LIN {X 0,Y 447.566,Z 552.365,A -85,B 0,C 180,E1 -8885.391,E2 -8885.391} C_VEL
LIN {X 0,Y 445.234,Z 544.551,A -85,B 0,C 180,E1 -8886.114,E2 -8886.114} C_VEL
LIN {X 0,Y 442.806,Z 536.367,A -85,B 0,C 180,E1 -8886.763,E2 -8886.763} C_VEL
LIN {X 0,Y 442.293,Z 531.074,A -85,B 0,C 180,E1 -8887.095,E2 -8887.095} C_VEL
LIN {X 0,Y 442.72,Z 518.254,A -85,B 0,C 180,E1 -8887.696,E2 -8887.696} C_VEL
LIN {X 0,Y 443.107,Z 504.32,A -85,B 0,C 180,E1 -8888.13,E2 -8888.13} C_VEL
LIN {X 0,Y 444.089,Z 414.582,A -85,B 0,C 180,E1 -8889.651,E2 -8889.651} C_VEL
LIN {X 0,Y 440.694,Z 396.943,A -85,B 0,C 180,E1 -8890.111,E2 -8890.111} C_VEL
LIN {X 0,Y 441.167,Z 386.817,A -85,B 0,C 180,E1 -8892.38,E2 -8892.38} C_VEL
LIN {X 0,Y 439.924,Z 378.992,A -85,B 0,C 180,E1 -8894.24,E2 -8894.24} C_VEL
LIN {X 0,Y 439.488,Z 376.743,A -85,B 0,C 180,E1 -8894.819,E2 -8894.819} C_VEL
LIN {X 0,Y 439.491,Z 376.739,A -85,B 0,C 180,E1 -8898,E2 -8898} C_VEL
LIN {X 0,Y 439.538,Z 376.73,A -85,B 0,C 180,E1 -8901.725,E2 -8901.725} C_VEL
LIN {X 0,Y 439.615,Z 376.728,A -85,B 0,C 180,E1 -8904.495,E2 -8904.495} C_VEL
LIN {X 0,Y 439.639,Z 376.722,A -85,B 0,C 180,E1 -8908.167,E2 -8908.167} C_VEL
LIN {X 0,Y 439.767,Z 376.705,A -85,B 0,C 180,E1 -8909.999,E2 -8909.999} C_VEL
LIN {X 0,Y 439.659,Z 376.717,A -85,B 0,C 180,E1 -8912.747,E2 -8912.747} C_VEL
LIN {X 0,Y 439.621,Z 376.724,A -85,B 0,C 180,E1 -8916.424,E2 -8916.424} C_VEL
LIN {X 0,Y 439.501,Z 376.734,A -85,B 0,C 180,E1 -8919.2,E2 -8919.2} C_VEL
LIN {X 0,Y 439.467,Z 376.739,A -85,B 0,C 180,E1 -8922.936,E2 -8922.936} C_VEL
LIN {X 0,Y 439.461,Z 376.743,A -85,B 0,C 180,E1 -8926.353,E2 -8926.353} C_VEL
LIN {X 0,Y 439.403,Z 376.75,A -85,B 0,C 180,E1 -8929.625,E2 -8929.625} C_VEL
LIN {X 0,Y 439.363,Z 376.753,A -85,B 0,C 180,E1 -8932.574,E2 -8932.574} C_VEL
LIN {X 0,Y 439.396,Z 376.752,A -85,B 0,C 180,E1 -8935.584,E2 -8935.584} C_VEL
LIN {X 0,Y 439.423,Z 376.744,A -85,B 0,C 180,E1 -8938.671,E2 -8938.671} C_VEL
LIN {X 0,Y 439.38,Z 376.753,A -85,B 0,C 180,E1 -8942.032,E2 -8942.032} C_VEL
LIN {X 0,Y 439.393,Z 376.752,A -85,B 0,C 180,E1 -8945.339,E2 -8945.339} C_VEL
LIN {X 0,Y 439.394,Z 376.748,A -85,B 0,C 180,E1 -8948.592,E2 -8948.592} C_VEL
LIN {X 0,Y 439.394,Z 376.752,A -85,B 0,C 180,E1 -8951.257,E2 -8951.257} C_VEL
LIN {X 0,Y 439.4,Z 376.751,A -85,B 0,C 180,E1 -8954.727,E2 -8954.727} C_VEL
LIN {X 0,Y 439.447,Z 376.896,A -85,B 0,C 180,E1 -8956.182,E2 -8956.182} C_VEL
LIN {X 0,Y 440.645,Z 383.573,A -85,B 0,C 180,E1 -8957.581,E2 -8957.581} C_VEL
LIN {X 0,Y 440.586,Z 391.432,A -85,B 0,C 180,E1 -8959.155,E2 -8959.155} C_VEL
LIN {X 0,Y 440.543,Z 396.061,A -85,B 0,C 180,E1 -8960.073,E2 -8960.073} C_VEL
LIN {X 0,Y 443.892,Z 415.086,A -85,B 0,C 180,E1 -8960.552,E2 -8960.552} C_VEL
LIN {X 0,Y 442.71,Z 504.451,A -85,B 0,C 180,E1 -8962.148,E2 -8962.148} C_VEL
LIN {X 0,Y 442.406,Z 517.033,A -85,B 0,C 180,E1 -8962.539,E2 -8962.539} C_VEL
LIN {X 0,Y 441.999,Z 529.5,A -85,B 0,C 180,E1 -8963.112,E2 -8963.112} C_VEL
LIN {X 0,Y 441.424,Z 542.347,A -85,B 0,C 180,E1 -8963.908,E2 -8963.908} C_VEL
LIN {X 0,Y 440.846,Z 554.105,A -85,B 0,C 180,E1 -8964.864,E2 -8964.864} C_VEL
LIN {X 0,Y 440.299,Z 564.276,A -85,B 0,C 180,E1 -8965.898,E2 -8965.898} C_VEL
LIN {X 0,Y 439.735,Z 573.76,A -85,B 0,C 180,E1 -8967.084,E2 -8967.084} C_VEL
LIN {X 0,Y 439.346,Z 582.271,A -85,B 0,C 180,E1 -8968.406,E2 -8968.406} C_VEL
LIN {X 0,Y 438.905,Z 589.744,A -85,B 0,C 180,E1 -8969.843,E2 -8969.843} C_VEL
LIN {X 0,Y 438.641,Z 595.595,A -85,B 0,C 180,E1 -8971.271,E2 -8971.271} C_VEL
LIN {X 0,Y 438.411,Z 600.454,A -85,B 0,C 180,E1 -8972.814,E2 -8972.814} C_VEL
LIN {X 0,Y 438.281,Z 603.953,A -85,B 0,C 180,E1 -8974.345,E2 -8974.345} C_VEL
LIN {X 0,Y 438.161,Z 606.47,A -85,B 0,C 180,E1 -8976.098,E2 -8976.098} C_VEL
LIN {X 0,Y 438.109,Z 607.349,A -85,B 0,C 180,E1 -8977.356,E2 -8977.356} C_VEL
LIN {X 0,Y 438.125,Z 607.446,A -85,B 0,C 180,E1 -8978.49,E2 -8978.49} C_VEL
LIN {X 0,Y 438.167,Z 607.132,A -85,B 0,C 180,E1 -8979.337,E2 -8979.337} C_VEL
LIN {X 0,Y 438.189,Z 606.343,A -85,B 0,C 180,E1 -8980.317,E2 -8980.317} C_VEL
LIN {X 0,Y 438.258,Z 605.052,A -85,B 0,C 180,E1 -8981.293,E2 -8981.293} C_VEL
LIN {X 0,Y 438.387,Z 602.262,A -85,B 0,C 180,E1 -8982.747,E2 -8982.747} C_VEL
LIN {X 0,Y 438.537,Z 598.37,A -85,B 0,C 180,E1 -8984.19,E2 -8984.19} C_VEL
LIN {X 0,Y 438.814,Z 593.262,A -85,B 0,C 180,E1 -8985.626,E2 -8985.626} C_VEL
LIN {X 0,Y 439.199,Z 586.765,A -85,B 0,C 180,E1 -8987.054,E2 -8987.054} C_VEL
LIN {X 0,Y 439.664,Z 578.655,A -85,B 0,C 180,E1 -8988.474,E2 -8988.474} C_VEL
LIN {X 0,Y 440.14,Z 570.383,A -85,B 0,C 180,E1 -8989.651,E2 -8989.651} C_VEL
LIN {X 0,Y 440.783,Z 560.176,A -85,B 0,C 180,E1 -8990.825,E2 -8990.825} C_VEL
LIN {X 0,Y 441.464,Z 548.726,A -85,B 0,C 180,E1 -8991.878,E2 -8991.878} C_VEL
LIN {X 0,Y 442.006,Z 537.482,A -85,B 0,C 180,E1 -8992.692,E2 -8992.692} C_VEL
LIN {X 0,Y 442.484,Z 524.938,A -85,B 0,C 180,E1 -8993.387,E2 -8993.387} C_VEL
LIN {X 0,Y 442.894,Z 511.882,A -85,B 0,C 180,E1 -8993.908,E2 -8993.908} C_VEL
LIN {X 0,Y 443.187,Z 497.848,A -85,B 0,C 180,E1 -8994.255,E2 -8994.255} C_VEL
LIN {X 0,Y 444.33,Z 414.224,A -85,B 0,C 180,E1 -8995.784,E2 -8995.784} C_VEL
LIN {X 0,Y 440.81,Z 396.654,A -85,B 0,C 180,E1 -8996.308,E2 -8996.308} C_VEL
LIN {X 0,Y 441.009,Z 384.795,A -85,B 0,C 180,E1 -8998.63,E2 -8998.63} C_VEL
LIN {X 0,Y 439.724,Z 376.714,A -85,B 0,C 180,E1 -9000.286,E2 -9000.286} C_VEL
LIN {X 0,Y 439.647,Z 376.725,A -85,B 0,C 180,E1 -9002.749,E2 -9002.749} C_VEL
LIN {X 0,Y 439.608,Z 376.728,A -85,B 0,C 180,E1 -9006.425,E2 -9006.425} C_VEL
LIN {X 0,Y 439.491,Z 376.739,A -85,B 0,C 180,E1 -9009.202,E2 -9009.202} C_VEL
LIN {X 0,Y 439.493,Z 376.741,A -85,B 0,C 180,E1 -9012.727,E2 -9012.727} C_VEL
LIN {X 0,Y 439.449,Z 376.747,A -85,B 0,C 180,E1 -9016.355,E2 -9016.355} C_VEL
LIN {X 0,Y 439.425,Z 376.75,A -85,B 0,C 180,E1 -9019.625,E2 -9019.625} C_VEL
LIN {X 0,Y 439.376,Z 376.752,A -85,B 0,C 180,E1 -9022.575,E2 -9022.575} C_VEL
LIN {X 0,Y 439.405,Z 376.753,A -85,B 0,C 180,E1 -9025.585,E2 -9025.585} C_VEL
LIN {X 0,Y 439.415,Z 376.747,A -85,B 0,C 180,E1 -9028.674,E2 -9028.674} C_VEL
LIN {X 0,Y 439.374,Z 376.755,A -85,B 0,C 180,E1 -9032.034,E2 -9032.034} C_VEL
LIN {X 0,Y 439.387,Z 376.754,A -85,B 0,C 180,E1 -9035.342,E2 -9035.342} C_VEL
LIN {X 0,Y 439.382,Z 376.751,A -85,B 0,C 180,E1 -9038.595,E2 -9038.595} C_VEL
LIN {X 0,Y 439.382,Z 376.755,A -85,B 0,C 180,E1 -9041.258,E2 -9041.258} C_VEL
LIN {X 0,Y 439.399,Z 376.75,A -85,B 0,C 180,E1 -9044.73,E2 -9044.73} C_VEL
LIN {X 0,Y 439.391,Z 376.751,A -85,B 0,C 180,E1 -9047.797,E2 -9047.797} C_VEL
LIN {X 0,Y 439.424,Z 376.746,A -85,B 0,C 180,E1 -9050.229,E2 -9050.229} C_VEL
LIN {X 0,Y 439.372,Z 376.753,A -85,B 0,C 180,E1 -9053.715,E2 -9053.715} C_VEL
LIN {X 0,Y 439.372,Z 376.758,A -85,B 0,C 180,E1 -9057.056,E2 -9057.056} C_VEL
LIN {X 0,Y 439.395,Z 376.753,A -85,B 0,C 180,E1 -9060.277,E2 -9060.277} C_VEL
LIN {X 0,Y 439.481,Z 376.95,A -85,B 0,C 180,E1 -9063.401,E2 -9063.401} C_VEL
LIN {X 0,Y 441.912,Z 389.672,A -85,B 0,C 180,E1 -9066.076,E2 -9066.076} C_VEL
LIN {X 0,Y 441.931,Z 394.416,A -85,B 0,C 180,E1 -9067.01,E2 -9067.01} C_VEL
LIN {X 0,Y 440.88,Z 413.613,A -85,B 0,C 180,E1 -9070.686,E2 -9070.686} C_VEL
LIN {X 0,Y 440.489,Z 420.151,A -85,B 0,C 180,E1 -9071.923,E2 -9071.923} C_VEL
LIN {X 0,Y 443.955,Z 442.221,A -85,B 0,C 180,E1 -9072.443,E2 -9072.443} C_VEL
LIN {X 0,Y 443.036,Z 528.918,A -85,B 0,C 180,E1 -9073.913,E2 -9073.913} C_VEL
LIN {X 0,Y 442.567,Z 542.639,A -85,B 0,C 180,E1 -9074.339,E2 -9074.339} C_VEL
LIN {X 0,Y 442.07,Z 555.017,A -85,B 0,C 180,E1 -9074.912,E2 -9074.912} C_VEL
LIN {X 0,Y 441.505,Z 566.099,A -85,B 0,C 180,E1 -9075.599,E2 -9075.599} C_VEL
LIN {X 0,Y 440.859,Z 577.655,A -85,B 0,C 180,E1 -9076.517,E2 -9076.517} C_VEL
LIN {X 0,Y 440.298,Z 588.106,A -85,B 0,C 180,E1 -9077.557,E2 -9077.557} C_VEL
LIN {X 0,Y 439.725,Z 597.48,A -85,B 0,C 180,E1 -9078.711,E2 -9078.711} C_VEL
LIN {X 0,Y 439.182,Z 606.551,A -85,B 0,C 180,E1 -9080.096,E2 -9080.096} C_VEL
LIN {X 0,Y 438.798,Z 613.859,A -85,B 0,C 180,E1 -9081.481,E2 -9081.481} C_VEL
LIN {X 0,Y 438.582,Z 618.796,A -85,B 0,C 180,E1 -9082.636,E2 -9082.636} C_VEL
LIN {X 0,Y 438.384,Z 623.457,A -85,B 0,C 180,E1 -9083.978,E2 -9083.978} C_VEL
LIN {X 0,Y 438.341,Z 627.253,A -85,B 0,C 180,E1 -9085.403,E2 -9085.403} C_VEL
LIN {X 0,Y 438.28,Z 629.143,A -85,B 0,C 180,E1 -9086.324,E2 -9086.324} C_VEL
LIN {X 0,Y 438.34,Z 630.568,A -85,B 0,C 180,E1 -9087.244,E2 -9087.244} C_VEL
LIN {X 0,Y 438.252,Z 632.191,A -85,B 0,C 180,E1 -9089.082,E2 -9089.082} C_VEL
LIN {X 0,Y 438.253,Z 632.415,A -85,B 0,C 180,E1 -9090.001,E2 -9090.001} C_VEL
LIN {X 0,Y 438.252,Z 632.202,A -85,B 0,C 180,E1 -9090.92,E2 -9090.92} C_VEL
LIN {X 0,Y 438.341,Z 630.585,A -85,B 0,C 180,E1 -9092.758,E2 -9092.758} C_VEL
LIN {X 0,Y 438.28,Z 629.174,A -85,B 0,C 180,E1 -9093.679,E2 -9093.679} C_VEL
LIN {X 0,Y 438.386,Z 626.213,A -85,B 0,C 180,E1 -9095.06,E2 -9095.06} C_VEL
LIN {X 0,Y 438.449,Z 622.202,A -85,B 0,C 180,E1 -9096.444,E2 -9096.444} C_VEL
LIN {X 0,Y 438.688,Z 616.038,A -85,B 0,C 180,E1 -9098.059,E2 -9098.059} C_VEL
LIN {X 0,Y 439.048,Z 609.304,A -85,B 0,C 180,E1 -9099.445,E2 -9099.445} C_VEL
LIN {X 0,Y 439.489,Z 600.961,A -85,B 0,C 180,E1 -9100.831,E2 -9100.831} C_VEL
LIN {X 0,Y 440.08,Z 592.405,A -85,B 0,C 180,E1 -9101.983,E2 -9101.983} C_VEL
LIN {X 0,Y 440.612,Z 582.48,A -85,B 0,C 180,E1 -9103.075,E2 -9103.075} C_VEL
LIN {X 0,Y 441.266,Z 571.393,A -85,B 0,C 180,E1 -9104.058,E2 -9104.058} C_VEL
LIN {X 0,Y 441.886,Z 559.936,A -85,B 0,C 180,E1 -9104.861,E2 -9104.861} C_VEL
LIN {X 0,Y 442.507,Z 548.123,A -85,B 0,C 180,E1 -9105.488,E2 -9105.488} C_VEL
LIN {X 0,Y 442.942,Z 535.462,A -85,B 0,C 180,E1 -9105.974,E2 -9105.974} C_VEL
LIN {X 0,Y 443.357,Z 522.565,A -85,B 0,C 180,E1 -9106.284,E2 -9106.284} C_VEL
LIN {X 0,Y 444.033,Z 441.38,A -85,B 0,C 180,E1 -9107.656,E2 -9107.656} C_VEL
LIN {X 0,Y 440.537,Z 419.596,A -85,B 0,C 180,E1 -9108.203,E2 -9108.203} C_VEL
LIN {X 0,Y 441.514,Z 402.491,A -85,B 0,C 180,E1 -9111.477,E2 -9111.477} C_VEL
LIN {X 0,Y 442.185,Z 391.264,A -85,B 0,C 180,E1 -9113.662,E2 -9113.662} C_VEL
LIN {X 0,Y 440.418,Z 381.325,A -85,B 0,C 180,E1 -9115.77,E2 -9115.77} C_VEL
LIN {X 0,Y 439.449,Z 376.748,A -85,B 0,C 180,E1 -9116.796,E2 -9116.796} C_VEL
LIN {X 0,Y 439.388,Z 376.757,A -85,B 0,C 180,E1 -9119.726,E2 -9119.726} C_VEL
LIN {X 0,Y 439.378,Z 376.757,A -85,B 0,C 180,E1 -9122.947,E2 -9122.947} C_VEL
LIN {X 0,Y 439.379,Z 376.754,A -85,B 0,C 180,E1 -9126.288,E2 -9126.288} C_VEL
LIN {X 0,Y 439.412,Z 376.751,A -85,B 0,C 180,E1 -9129.85,E2 -9129.85} C_VEL
LIN {X 0,Y 439.388,Z 376.755,A -85,B 0,C 180,E1 -9132.628,E2 -9132.628} C_VEL
LIN {X 0,Y 439.407,Z 376.753,A -85,B 0,C 180,E1 -9135.271,E2 -9135.271} C_VEL
LIN {X 0,Y 439.394,Z 376.755,A -85,B 0,C 180,E1 -9138.744,E2 -9138.744} C_VEL
LIN {X 0,Y 439.378,Z 376.752,A -85,B 0,C 180,E1 -9141.608,E2 -9141.608} C_VEL
LIN {X 0,Y 439.404,Z 376.752,A -85,B 0,C 180,E1 -9144.844,E2 -9144.844} C_VEL
LIN {X 0,Y 439.379,Z 376.752,A -85,B 0,C 180,E1 -9148.14,E2 -9148.14} C_VEL
LIN {X 0,Y 439.438,Z 376.743,A -85,B 0,C 180,E1 -9151.598,E2 -9151.598} C_VEL
LIN {X 0,Y 439.403,Z 376.749,A -85,B 0,C 180,E1 -9154.415,E2 -9154.415} C_VEL
LIN {X 0,Y 439.369,Z 376.747,A -85,B 0,C 180,E1 -9157.425,E2 -9157.425} C_VEL
LIN {X 0,Y 439.447,Z 376.742,A -85,B 0,C 180,E1 -9160.663,E2 -9160.663} C_VEL
LIN {X 0,Y 439.468,Z 376.745,A -85,B 0,C 180,E1 -9164.225,E2 -9164.225} C_VEL
LIN {X 0,Y 439.489,Z 376.741,A -85,B 0,C 180,E1 -9168.001,E2 -9168.001} C_VEL
LIN {X 0,Y 439.554,Z 376.731,A -85,B 0,C 180,E1 -9171.726,E2 -9171.726} C_VEL
LIN {X 0,Y 439.627,Z 376.724,A -85,B 0,C 180,E1 -9174.496,E2 -9174.496} C_VEL
LIN {X 0,Y 439.64,Z 376.723,A -85,B 0,C 180,E1 -9178.168,E2 -9178.168} C_VEL
LIN {X 0,Y 439.768,Z 376.706,A -85,B 0,C 180,E1 -9180,E2 -9180} C_VEL
LIN {X 0,Y 439.647,Z 376.718,A -85,B 0,C 180,E1 -9182.749,E2 -9182.749} C_VEL
LIN {X 0,Y 439.624,Z 376.721,A -85,B 0,C 180,E1 -9186.425,E2 -9186.425} C_VEL
LIN {X 0,Y 439.506,Z 376.736,A -85,B 0,C 180,E1 -9189.202,E2 -9189.202} C_VEL
LIN {X 0,Y 439.472,Z 376.74,A -85,B 0,C 180,E1 -9192.938,E2 -9192.938} C_VEL
LIN {X 0,Y 439.454,Z 376.744,A -85,B 0,C 180,E1 -9196.349,E2 -9196.349} C_VEL
LIN {X 0,Y 439.409,Z 376.753,A -85,B 0,C 180,E1 -9199.626,E2 -9199.626} C_VEL
LIN {X 0,Y 439.37,Z 376.754,A -85,B 0,C 180,E1 -9202.575,E2 -9202.575} C_VEL
LIN {X 0,Y 439.404,Z 376.752,A -85,B 0,C 180,E1 -9205.585,E2 -9205.585} C_VEL
LIN {X 0,Y 439.461,Z 376.78,A -85,B 0,C 180,E1 -9208.965,E2 -9208.965} C_VEL
LIN {X 0,Y 441.273,Z 386.843,A -85,B 0,C 180,E1 -9211.44,E2 -9211.44} C_VEL
LIN {X 0,Y 440.869,Z 397.525,A -85,B 0,C 180,E1 -9213.88,E2 -9213.88} C_VEL
LIN {X 0,Y 444.38,Z 415.736,A -85,B 0,C 180,E1 -9214.365,E2 -9214.365} C_VEL
LIN {X 0,Y 443.296,Z 504.669,A -85,B 0,C 180,E1 -9215.881,E2 -9215.881} C_VEL
LIN {X 0,Y 442.938,Z 517.91,A -85,B 0,C 180,E1 -9216.292,E2 -9216.292} C_VEL
LIN {X 0,Y 442.511,Z 529.911,A -85,B 0,C 180,E1 -9216.841,E2 -9216.841} C_VEL
LIN {X 0,Y 441.995,Z 541.351,A -85,B 0,C 180,E1 -9217.54,E2 -9217.54} C_VEL
LIN {X 0,Y 441.402,Z 552.126,A -85,B 0,C 180,E1 -9218.386,E2 -9218.386} C_VEL
LIN {X 0,Y 440.719,Z 563.511,A -85,B 0,C 180,E1 -9219.51,E2 -9219.51} C_VEL
LIN {X 0,Y 440.06,Z 572.934,A -85,B 0,C 180,E1 -9220.669,E2 -9220.669} C_VEL
LIN {X 0,Y 439.57,Z 581.346,A -85,B 0,C 180,E1 -9221.953,E2 -9221.953} C_VEL
LIN {X 0,Y 439.166,Z 587.526,A -85,B 0,C 180,E1 -9223.092,E2 -9223.092} C_VEL
LIN {X 0,Y 438.861,Z 593.327,A -85,B 0,C 180,E1 -9224.396,E2 -9224.396} C_VEL
LIN {X 0,Y 438.613,Z 598.01,A -85,B 0,C 180,E1 -9225.702,E2 -9225.702} C_VEL
LIN {X 0,Y 438.42,Z 601.693,A -85,B 0,C 180,E1 -9227.008,E2 -9227.008} C_VEL
LIN {X 0,Y 438.296,Z 604.387,A -85,B 0,C 180,E1 -9228.282,E2 -9228.282} C_VEL
LIN {X 0,Y 438.142,Z 606.786,A -85,B 0,C 180,E1 -9230.086,E2 -9230.086} C_VEL
LIN {X 0,Y 438.137,Z 607.642,A -85,B 0,C 180,E1 -9231.813,E2 -9231.813} C_VEL
LIN {X 0,Y 438.152,Z 607.06,A -85,B 0,C 180,E1 -9233.594,E2 -9233.594} C_VEL
LIN {X 0,Y 438.2,Z 605.696,A -85,B 0,C 180,E1 -9234.881,E2 -9234.881} C_VEL
LIN {X 0,Y 438.389,Z 602.878,A -85,B 0,C 180,E1 -9236.474,E2 -9236.474} C_VEL
LIN {X 0,Y 438.561,Z 598.488,A -85,B 0,C 180,E1 -9238.14,E2 -9238.14} C_VEL
LIN {X 0,Y 438.79,Z 593.541,A -85,B 0,C 180,E1 -9239.545,E2 -9239.545} C_VEL
LIN {X 0,Y 439.21,Z 586.801,A -85,B 0,C 180,E1 -9241.049,E2 -9241.049} C_VEL
LIN {X 0,Y 439.654,Z 579.288,A -85,B 0,C 180,E1 -9242.381,E2 -9242.381} C_VEL
LIN {X 0,Y 440.169,Z 570.074,A -85,B 0,C 180,E1 -9243.699,E2 -9243.699} C_VEL
LIN {X 0,Y 440.769,Z 560.449,A -85,B 0,C 180,E1 -9244.815,E2 -9244.815} C_VEL
LIN {X 0,Y 441.379,Z 550,A -85,B 0,C 180,E1 -9245.793,E2 -9245.793} C_VEL
LIN {X 0,Y 441.991,Z 538.279,A -85,B 0,C 180,E1 -9246.659,E2 -9246.659} C_VEL
LIN {X 0,Y 442.293,Z 531.074,A -85,B 0,C 180,E1 -9247.095,E2 -9247.095} C_VEL
LIN {X 0,Y 441.795,Z 525.662,A -85,B 0,C 180,E1 -9247.399,E2 -9247.399} C_VEL
LIN {X 0,Y 439.368,Z 516.782,A -85,B 0,C 180,E1 -9247.88,E2 -9247.88} C_VEL
LIN {X 0,Y 436.901,Z 507.688,A -85,B 0,C 180,E1 -9248.27,E2 -9248.27} C_VEL
LIN {X 0,Y 436.322,Z 501.949,A -85,B 0,C 180,E1 -9248.427,E2 -9248.427} C_VEL
LIN {X 0,Y 437.208,Z 415.029,A -85,B 0,C 180,E1 -9249.919,E2 -9249.919} C_VEL
LIN {X 0,Y 433.767,Z 397.177,A -85,B 0,C 180,E1 -9250.384,E2 -9250.384} C_VEL
LIN {X 0,Y 434.141,Z 387.363,A -85,B 0,C 180,E1 -9252.621,E2 -9252.621} C_VEL
LIN {X 0,Y 432.459,Z 377.619,A -85,B 0,C 180,E1 -9255.018,E2 -9255.018} C_VEL
LIN {X 0,Y 432.464,Z 377.614,A -85,B 0,C 180,E1 -9257.802,E2 -9257.802} C_VEL
LIN {X 0,Y 432.488,Z 377.608,A -85,B 0,C 180,E1 -9261.589,E2 -9261.589} C_VEL
LIN {X 0,Y 432.59,Z 377.603,A -85,B 0,C 180,E1 -9264.405,E2 -9264.405} C_VEL
LIN {X 0,Y 432.609,Z 377.598,A -85,B 0,C 180,E1 -9268.137,E2 -9268.137} C_VEL
LIN {X 0,Y 432.736,Z 377.581,A -85,B 0,C 180,E1 -9269.999,E2 -9269.999} C_VEL
LIN {X 0,Y 432.608,Z 377.595,A -85,B 0,C 180,E1 -9272.792,E2 -9272.792} C_VEL
LIN {X 0,Y 432.576,Z 377.601,A -85,B 0,C 180,E1 -9276.529,E2 -9276.529} C_VEL
LIN {X 0,Y 432.444,Z 377.614,A -85,B 0,C 180,E1 -9279.352,E2 -9279.352} C_VEL
LIN {X 0,Y 432.432,Z 377.616,A -85,B 0,C 180,E1 -9282.802,E2 -9282.802} C_VEL
LIN {X 0,Y 432.424,Z 377.618,A -85,B 0,C 180,E1 -9286.482,E2 -9286.482} C_VEL
LIN {X 0,Y 432.339,Z 377.634,A -85,B 0,C 180,E1 -9289.959,E2 -9289.959} C_VEL
LIN {X 0,Y 432.317,Z 377.63,A -85,B 0,C 180,E1 -9292.963,E2 -9292.963} C_VEL
LIN {X 0,Y 432.36,Z 377.629,A -85,B 0,C 180,E1 -9296.031,E2 -9296.031} C_VEL
LIN {X 0,Y 432.35,Z 377.627,A -85,B 0,C 180,E1 -9299.185,E2 -9299.185} C_VEL
LIN {X 0,Y 432.329,Z 377.629,A -85,B 0,C 180,E1 -9302.293,E2 -9302.293} C_VEL
LIN {X 0,Y 432.337,Z 377.627,A -85,B 0,C 180,E1 -9304.675,E2 -9304.675} C_VEL
LIN {X 0,Y 432.348,Z 377.627,A -85,B 0,C 180,E1 -9308.147,E2 -9308.147} C_VEL
LIN {X 0,Y 432.362,Z 377.631,A -85,B 0,C 180,E1 -9311.606,E2 -9311.606} C_VEL
LIN {X 0,Y 432.335,Z 377.631,A -85,B 0,C 180,E1 -9314.345,E2 -9314.345} C_VEL
LIN {X 0,Y 432.39,Z 377.751,A -85,B 0,C 180,E1 -9316.031,E2 -9316.031} C_VEL
LIN {X 0,Y 433.737,Z 385.68,A -85,B 0,C 180,E1 -9317.693,E2 -9317.693} C_VEL
LIN {X 0,Y 433.561,Z 396.365,A -85,B 0,C 180,E1 -9319.806,E2 -9319.806} C_VEL
LIN {X 0,Y 437.065,Z 415.855,A -85,B 0,C 180,E1 -9320.314,E2 -9320.314} C_VEL
LIN {X 0,Y 435.859,Z 503.979,A -85,B 0,C 180,E1 -9321.92,E2 -9321.92} C_VEL
LIN {X 0,Y 435.5,Z 517.172,A -85,B 0,C 180,E1 -9322.331,E2 -9322.331} C_VEL
LIN {X 0,Y 435.055,Z 529.986,A -85,B 0,C 180,E1 -9322.932,E2 -9322.932} C_VEL
LIN {X 0,Y 434.481,Z 542.469,A -85,B 0,C 180,E1 -9323.719,E2 -9323.719} C_VEL
LIN {X 0,Y 433.929,Z 553.476,A -85,B 0,C 180,E1 -9324.618,E2 -9324.618} C_VEL
LIN {X 0,Y 433.321,Z 563.929,A -85,B 0,C 180,E1 -9325.683,E2 -9325.683} C_VEL
LIN {X 0,Y 432.81,Z 572.642,A -85,B 0,C 180,E1 -9326.767,E2 -9326.767} C_VEL
LIN {X 0,Y 432.355,Z 581.436,A -85,B 0,C 180,E1 -9328.11,E2 -9328.11} C_VEL
LIN {X 0,Y 431.872,Z 589.21,A -85,B 0,C 180,E1 -9329.594,E2 -9329.594} C_VEL
LIN {X 0,Y 431.642,Z 594.154,A -85,B 0,C 180,E1 -9330.76,E2 -9330.76} C_VEL
LIN {X 0,Y 431.406,Z 599.473,A -85,B 0,C 180,E1 -9332.335,E2 -9332.335} C_VEL
LIN {X 0,Y 431.24,Z 603.332,A -85,B 0,C 180,E1 -9333.894,E2 -9333.894} C_VEL
LIN {X 0,Y 431.142,Z 605.168,A -85,B 0,C 180,E1 -9334.924,E2 -9334.924} C_VEL
LIN {X 0,Y 431.076,Z 606.522,A -85,B 0,C 180,E1 -9335.947,E2 -9335.947} C_VEL
LIN {X 0,Y 431.018,Z 607.322,A -85,B 0,C 180,E1 -9336.962,E2 -9336.962} C_VEL
LIN {X 0,Y 431.024,Z 607.665,A -85,B 0,C 180,E1 -9338.338,E2 -9338.338} C_VEL
LIN {X 0,Y 431.098,Z 606.895,A -85,B 0,C 180,E1 -9339.98,E2 -9339.98} C_VEL
LIN {X 0,Y 431.138,Z 605.819,A -85,B 0,C 180,E1 -9340.985,E2 -9340.985} C_VEL
LIN {X 0,Y 431.264,Z 603.331,A -85,B 0,C 180,E1 -9342.453,E2 -9342.453} C_VEL
LIN {X 0,Y 431.438,Z 599.618,A -85,B 0,C 180,E1 -9343.958,E2 -9343.958} C_VEL
LIN {X 0,Y 431.681,Z 594.924,A -85,B 0,C 180,E1 -9345.383,E2 -9345.383} C_VEL
LIN {X 0,Y 432.046,Z 588.803,A -85,B 0,C 180,E1 -9346.836,E2 -9346.836} C_VEL
LIN {X 0,Y 432.578,Z 581.157,A -85,B 0,C 180,E1 -9348.282,E2 -9348.282} C_VEL
LIN {X 0,Y 433.031,Z 573.341,A -85,B 0,C 180,E1 -9349.479,E2 -9349.479} C_VEL
LIN {X 0,Y 433.64,Z 563.788,A -85,B 0,C 180,E1 -9350.673,E2 -9350.673} C_VEL
LIN {X 0,Y 434.314,Z 553.251,A -85,B 0,C 180,E1 -9351.743,E2 -9351.743} C_VEL
LIN {X 0,Y 434.962,Z 541.428,A -85,B 0,C 180,E1 -9352.69,E2 -9352.69} C_VEL
LIN {X 0,Y 435.547,Z 529.049,A -85,B 0,C 180,E1 -9353.456,E2 -9353.456} C_VEL
LIN {X 0,Y 435.992,Z 516.01,A -85,B 0,C 180,E1 -9354.044,E2 -9354.044} C_VEL
LIN {X 0,Y 436.355,Z 502.175,A -85,B 0,C 180,E1 -9354.454,E2 -9354.454} C_VEL
LIN {X 0,Y 437.674,Z 415.448,A -85,B 0,C 180,E1 -9356.08,E2 -9356.08} C_VEL
LIN {X 0,Y 434.197,Z 398.146,A -85,B 0,C 180,E1 -9356.607,E2 -9356.607} C_VEL
LIN {X 0,Y 433.92,Z 396.665,A -85,B 0,C 180,E1 -9356.692,E2 -9356.692} C_VEL
LIN {X 0,Y 434.147,Z 386.949,A -85,B 0,C 180,E1 -9358.609,E2 -9358.609} C_VEL
LIN {X 0,Y 432.958,Z 379.029,A -85,B 0,C 180,E1 -9360.232,E2 -9360.232} C_VEL
LIN {X 0,Y 432.663,Z 377.594,A -85,B 0,C 180,E1 -9360.582,E2 -9360.582} C_VEL
LIN {X 0,Y 432.596,Z 377.603,A -85,B 0,C 180,E1 -9362.794,E2 -9362.794} C_VEL
LIN {X 0,Y 432.562,Z 377.605,A -85,B 0,C 180,E1 -9366.53,E2 -9366.53} C_VEL
LIN {X 0,Y 432.434,Z 377.618,A -85,B 0,C 180,E1 -9369.353,E2 -9369.353} C_VEL
LIN {X 0,Y 432.434,Z 377.62,A -85,B 0,C 180,E1 -9372.812,E2 -9372.812} C_VEL
LIN {X 0,Y 432.412,Z 377.623,A -85,B 0,C 180,E1 -9376.484,E2 -9376.484} C_VEL
LIN {X 0,Y 432.372,Z 377.629,A -85,B 0,C 180,E1 -9379.959,E2 -9379.959} C_VEL
LIN {X 0,Y 432.325,Z 377.629,A -85,B 0,C 180,E1 -9382.964,E2 -9382.964} C_VEL
LIN {X 0,Y 432.359,Z 377.629,A -85,B 0,C 180,E1 -9386.033,E2 -9386.033} C_VEL
LIN {X 0,Y 432.343,Z 377.63,A -85,B 0,C 180,E1 -9389.188,E2 -9389.188} C_VEL
LIN {X 0,Y 432.323,Z 377.632,A -85,B 0,C 180,E1 -9392.296,E2 -9392.296} C_VEL
LIN {X 0,Y 432.332,Z 377.63,A -85,B 0,C 180,E1 -9394.678,E2 -9394.678} C_VEL
LIN {X 0,Y 432.339,Z 377.629,A -85,B 0,C 180,E1 -9398.15,E2 -9398.15} C_VEL
LIN {X 0,Y 432.327,Z 377.634,A -85,B 0,C 180,E1 -9401.603,E2 -9401.603} C_VEL
LIN {X 0,Y 432.334,Z 377.628,A -85,B 0,C 180,E1 -9404.347,E2 -9404.347} C_VEL
LIN {X 0,Y 432.318,Z 377.636,A -85,B 0,C 180,E1 -9407.016,E2 -9407.016} C_VEL
LIN {X 0,Y 432.331,Z 377.63,A -85,B 0,C 180,E1 -9409.821,E2 -9409.821} C_VEL
LIN {X 0,Y 432.311,Z 377.638,A -85,B 0,C 180,E1 -9413.024,E2 -9413.024} C_VEL
LIN {X 0,Y 432.355,Z 377.628,A -85,B 0,C 180,E1 -9415.998,E2 -9415.998} C_VEL
LIN {X 0,Y 432.393,Z 377.624,A -85,B 0,C 180,E1 -9419.746,E2 -9419.746} C_VEL
LIN {X 0,Y 432.452,Z 377.635,A -85,B 0,C 180,E1 -9423.131,E2 -9423.131} C_VEL
LIN {X 0,Y 434.921,Z 390.685,A -85,B 0,C 180,E1 -9425.921,E2 -9425.921} C_VEL
LIN {X 0,Y 435.034,Z 394.74,A -85,B 0,C 180,E1 -9426.736,E2 -9426.736} C_VEL
LIN {X 0,Y 434.051,Z 410.991,A -85,B 0,C 180,E1 -9429.904,E2 -9429.904} C_VEL
LIN {X 0,Y 433.573,Z 419.896,A -85,B 0,C 180,E1 -9431.624,E2 -9431.624} C_VEL
LIN {X 0,Y 437.137,Z 443.181,A -85,B 0,C 180,E1 -9432.193,E2 -9432.193} C_VEL
LIN {X 0,Y 436.214,Z 528.054,A -85,B 0,C 180,E1 -9433.655,E2 -9433.655} C_VEL
LIN {X 0,Y 435.723,Z 541.231,A -85,B 0,C 180,E1 -9434.057,E2 -9434.057} C_VEL
LIN {X 0,Y 435.201,Z 554.51,A -85,B 0,C 180,E1 -9434.668,E2 -9434.668} C_VEL
LIN {X 0,Y 434.6,Z 565.677,A -85,B 0,C 180,E1 -9435.366,E2 -9435.366} C_VEL
LIN {X 0,Y 433.9,Z 577.507,A -85,B 0,C 180,E1 -9436.318,E2 -9436.318} C_VEL
LIN {X 0,Y 433.301,Z 587.77,A -85,B 0,C 180,E1 -9437.353,E2 -9437.353} C_VEL
LIN {X 0,Y 432.748,Z 597.187,A -85,B 0,C 180,E1 -9438.526,E2 -9438.526} C_VEL
LIN {X 0,Y 432.155,Z 606.28,A -85,B 0,C 180,E1 -9439.933,E2 -9439.933} C_VEL
LIN {X 0,Y 431.736,Z 613.605,A -85,B 0,C 180,E1 -9441.341,E2 -9441.341} C_VEL
LIN {X 0,Y 431.516,Z 618.557,A -85,B 0,C 180,E1 -9442.515,E2 -9442.515} C_VEL
LIN {X 0,Y 431.283,Z 623.662,A -85,B 0,C 180,E1 -9444.02,E2 -9444.02} C_VEL
LIN {X 0,Y 431.271,Z 627.033,A -85,B 0,C 180,E1 -9445.328,E2 -9445.328} C_VEL
LIN {X 0,Y 431.187,Z 628.927,A -85,B 0,C 180,E1 -9446.263,E2 -9446.263} C_VEL
LIN {X 0,Y 431.235,Z 630.358,A -85,B 0,C 180,E1 -9447.199,E2 -9447.199} C_VEL
LIN {X 0,Y 431.202,Z 631.369,A -85,B 0,C 180,E1 -9448.133,E2 -9448.133} C_VEL
LIN {X 0,Y 431.167,Z 632.214,A -85,B 0,C 180,E1 -9450.001,E2 -9450.001} C_VEL
LIN {X 0,Y 431.169,Z 632.005,A -85,B 0,C 180,E1 -9450.935,E2 -9450.935} C_VEL
LIN {X 0,Y 431.203,Z 631.393,A -85,B 0,C 180,E1 -9451.869,E2 -9451.869} C_VEL
LIN {X 0,Y 431.236,Z 630.389,A -85,B 0,C 180,E1 -9452.804,E2 -9452.804} C_VEL
LIN {X 0,Y 431.187,Z 628.982,A -85,B 0,C 180,E1 -9453.739,E2 -9453.739} C_VEL
LIN {X 0,Y 431.297,Z 626.023,A -85,B 0,C 180,E1 -9455.143,E2 -9455.143} C_VEL
LIN {X 0,Y 431.378,Z 622.019,A -85,B 0,C 180,E1 -9456.55,E2 -9456.55} C_VEL
LIN {X 0,Y 431.629,Z 615.866,A -85,B 0,C 180,E1 -9458.192,E2 -9458.192} C_VEL
LIN {X 0,Y 431.993,Z 609.143,A -85,B 0,C 180,E1 -9459.6,E2 -9459.6} C_VEL
LIN {X 0,Y 432.497,Z 600.806,A -85,B 0,C 180,E1 -9461.008,E2 -9461.008} C_VEL
LIN {X 0,Y 433.124,Z 592.262,A -85,B 0,C 180,E1 -9462.179,E2 -9462.179} C_VEL
LIN {X 0,Y 433.74,Z 581.416,A -85,B 0,C 180,E1 -9463.381,E2 -9463.381} C_VEL
LIN {X 0,Y 434.446,Z 569.84,A -85,B 0,C 180,E1 -9464.403,E2 -9464.403} C_VEL
LIN {X 0,Y 435.147,Z 557.892,A -85,B 0,C 180,E1 -9465.217,E2 -9465.217} C_VEL
LIN {X 0,Y 435.721,Z 545.49,A -85,B 0,C 180,E1 -9465.856,E2 -9465.856} C_VEL
LIN {X 0,Y 436.255,Z 532.756,A -85,B 0,C 180,E1 -9466.316,E2 -9466.316} C_VEL
LIN {X 0,Y 436.643,Z 517.724,A -85,B 0,C 180,E1 -9466.632,E2 -9466.632} C_VEL
LIN {X 0,Y 437.337,Z 442.517,A -85,B 0,C 180,E1 -9467.924,E2 -9467.924} C_VEL
LIN {X 0,Y 433.627,Z 419.336,A -85,B 0,C 180,E1 -9468.529,E2 -9468.529} C_VEL
LIN {X 0,Y 434.719,Z 401.143,A -85,B 0,C 180,E1 -9472.08,E2 -9472.08} C_VEL
LIN {X 0,Y 435.26,Z 392.429,A -85,B 0,C 180,E1 -9473.809,E2 -9473.809} C_VEL
LIN {X 0,Y 433.078,Z 380.821,A -85,B 0,C 180,E1 -9476.336,E2 -9476.336} C_VEL
LIN {X 0,Y 432.428,Z 377.624,A -85,B 0,C 180,E1 -9477.07,E2 -9477.07} C_VEL
LIN {X 0,Y 432.353,Z 377.63,A -85,B 0,C 180,E1 -9480.511,E2 -9480.511} C_VEL
LIN {X 0,Y 432.365,Z 377.626,A -85,B 0,C 180,E1 -9484.004,E2 -9484.004} C_VEL
LIN {X 0,Y 432.328,Z 377.637,A -85,B 0,C 180,E1 -9487.198,E2 -9487.198} C_VEL
LIN {X 0,Y 432.342,Z 377.631,A -85,B 0,C 180,E1 -9490.18,E2 -9490.18} C_VEL
LIN {X 0,Y 432.323,Z 377.637,A -85,B 0,C 180,E1 -9493.061,E2 -9493.061} C_VEL
LIN {X 0,Y 432.339,Z 377.63,A -85,B 0,C 180,E1 -9495.665,E2 -9495.665} C_VEL
LIN {X 0,Y 432.338,Z 377.63,A -85,B 0,C 180,E1 -9498.399,E2 -9498.399} C_VEL
LIN {X 0,Y 432.341,Z 377.628,A -85,B 0,C 180,E1 -9501.85,E2 -9501.85} C_VEL
LIN {X 0,Y 432.345,Z 377.626,A -85,B 0,C 180,E1 -9505.323,E2 -9505.323} C_VEL
LIN {X 0,Y 432.327,Z 377.633,A -85,B 0,C 180,E1 -9508.654,E2 -9508.654} C_VEL
LIN {X 0,Y 432.387,Z 377.622,A -85,B 0,C 180,E1 -9511.877,E2 -9511.877} C_VEL
LIN {X 0,Y 432.352,Z 377.629,A -85,B 0,C 180,E1 -9514.999,E2 -9514.999} C_VEL
LIN {X 0,Y 432.363,Z 377.622,A -85,B 0,C 180,E1 -9518.046,E2 -9518.046} C_VEL
LIN {X 0,Y 432.392,Z 377.617,A -85,B 0,C 180,E1 -9521.03,E2 -9521.03} C_VEL
LIN {X 0,Y 432.437,Z 377.618,A -85,B 0,C 180,E1 -9523.961,E2 -9523.961} C_VEL
LIN {X 0,Y 432.465,Z 377.614,A -85,B 0,C 180,E1 -9527.804,E2 -9527.804} C_VEL
LIN {X 0,Y 432.498,Z 377.609,A -85,B 0,C 180,E1 -9531.59,E2 -9531.59} C_VEL
LIN {X 0,Y 432.603,Z 377.6,A -85,B 0,C 180,E1 -9534.406,E2 -9534.406} C_VEL
LIN {X 0,Y 432.61,Z 377.598,A -85,B 0,C 180,E1 -9538.138,E2 -9538.138} C_VEL
LIN {X 0,Y 432.738,Z 377.581,A -85,B 0,C 180,E1 -9540,E2 -9540} C_VEL
LIN {X 0,Y 432.598,Z 377.596,A -85,B 0,C 180,E1 -9542.794,E2 -9542.794} C_VEL
LIN {X 0,Y 432.579,Z 377.598,A -85,B 0,C 180,E1 -9546.53,E2 -9546.53} C_VEL
LIN {X 0,Y 432.449,Z 377.617,A -85,B 0,C 180,E1 -9549.353,E2 -9549.353} C_VEL
LIN {X 0,Y 432.437,Z 377.617,A -85,B 0,C 180,E1 -9552.803,E2 -9552.803} C_VEL
LIN {X 0,Y 432.419,Z 377.62,A -85,B 0,C 180,E1 -9556.479,E2 -9556.479} C_VEL
LIN {X 0,Y 432.345,Z 377.633,A -85,B 0,C 180,E1 -9559.96,E2 -9559.96} C_VEL
LIN {X 0,Y 432.324,Z 377.633,A -85,B 0,C 180,E1 -9562.964,E2 -9562.964} C_VEL
LIN {X 0,Y 432.367,Z 377.63,A -85,B 0,C 180,E1 -9566.032,E2 -9566.032} C_VEL
LIN {X 0,Y 432.444,Z 377.665,A -85,B 0,C 180,E1 -9568.703,E2 -9568.703} C_VEL
LIN {X 0,Y 434.372,Z 388.649,A -85,B 0,C 180,E1 -9571.453,E2 -9571.453} C_VEL
LIN {X 0,Y 433.985,Z 397.685,A -85,B 0,C 180,E1 -9573.546,E2 -9573.546} C_VEL
LIN {X 0,Y 437.597,Z 415.604,A -85,B 0,C 180,E1 -9574.06,E2 -9574.06} C_VEL
LIN {X 0,Y 436.504,Z 505.056,A -85,B 0,C 180,E1 -9575.619,E2 -9575.619} C_VEL
LIN {X 0,Y 436.118,Z 518.507,A -85,B 0,C 180,E1 -9576.047,E2 -9576.047} C_VEL
LIN {X 0,Y 435.659,Z 531.191,A -85,B 0,C 180,E1 -9576.647,E2 -9576.647} C_VEL
LIN {X 0,Y 435.097,Z 542.438,A -85,B 0,C 180,E1 -9577.364,E2 -9577.364} C_VEL
LIN {X 0,Y 434.47,Z 553.064,A -85,B 0,C 180,E1 -9578.224,E2 -9578.224} C_VEL
LIN {X 0,Y 433.777,Z 564.079,A -85,B 0,C 180,E1 -9579.339,E2 -9579.339} C_VEL
LIN {X 0,Y 433.109,Z 573.115,A -85,B 0,C 180,E1 -9580.472,E2 -9580.472} C_VEL
LIN {X 0,Y 432.567,Z 581.498,A -85,B 0,C 180,E1 -9581.77,E2 -9581.77} C_VEL
LIN {X 0,Y 432.112,Z 588.443,A -85,B 0,C 180,E1 -9583.087,E2 -9583.087} C_VEL
LIN {X 0,Y 431.715,Z 595.233,A -85,B 0,C 180,E1 -9584.703,E2 -9584.703} C_VEL
LIN {X 0,Y 431.435,Z 600.305,A -85,B 0,C 180,E1 -9586.301,E2 -9586.301} C_VEL
LIN {X 0,Y 431.222,Z 604.322,A -85,B 0,C 180,E1 -9588.07,E2 -9588.07} C_VEL
LIN {X 0,Y 431.108,Z 606.198,A -85,B 0,C 180,E1 -9589.3,E2 -9589.3} C_VEL
LIN {X 0,Y 431.035,Z 607.377,A -85,B 0,C 180,E1 -9590.513,E2 -9590.513} C_VEL
LIN {X 0,Y 431.056,Z 607.829,A -85,B 0,C 180,E1 -9591.715,E2 -9591.715} C_VEL
LIN {X 0,Y 431.036,Z 607.599,A -85,B 0,C 180,E1 -9593.029,E2 -9593.029} C_VEL
LIN {X 0,Y 431.095,Z 606.279,A -85,B 0,C 180,E1 -9594.601,E2 -9594.601} C_VEL
LIN {X 0,Y 431.275,Z 603.455,A -85,B 0,C 180,E1 -9596.353,E2 -9596.353} C_VEL
LIN {X 0,Y 431.478,Z 599.718,A -85,B 0,C 180,E1 -9597.886,E2 -9597.886} C_VEL
LIN {X 0,Y 431.669,Z 595.656,A -85,B 0,C 180,E1 -9599.146,E2 -9599.146} C_VEL
LIN {X 0,Y 431.986,Z 590.137,A -85,B 0,C 180,E1 -9600.518,E2 -9600.518} C_VEL
LIN {X 0,Y 432.392,Z 583.348,A -85,B 0,C 180,E1 -9601.876,E2 -9601.876} C_VEL
LIN {X 0,Y 432.974,Z 574.292,A -85,B 0,C 180,E1 -9603.322,E2 -9603.322} C_VEL
LIN {X 0,Y 433.564,Z 564.691,A -85,B 0,C 180,E1 -9604.559,E2 -9604.559} C_VEL
LIN {X 0,Y 434.226,Z 554.392,A -85,B 0,C 180,E1 -9605.623,E2 -9605.623} C_VEL
LIN {X 0,Y 434.849,Z 542.221,A -85,B 0,C 180,E1 -9606.622,E2 -9606.622} C_VEL
LIN {X 0,Y 435.427,Z 529.904,A -85,B 0,C 180,E1 -9607.396,E2 -9607.396} C_VEL
LIN {X 0,Y 435.918,Z 516.633,A -85,B 0,C 180,E1 -9608,E2 -9608} C_VEL
LIN {X 0,Y 436.279,Z 504.091,A -85,B 0,C 180,E1 -9608.382,E2 -9608.382} C_VEL
LIN {X 0,Y 436.322,Z 501.949,A -85,B 0,C 180,E1 -9608.427,E2 -9608.427} C_VEL
LIN {X 0,Y 435.699,Z 496.158,A -85,B 0,C 180,E1 -9608.564,E2 -9608.564} C_VEL
LIN {X 0,Y 430.392,Z 477.466,A -85,B 0,C 180,E1 -9609.089,E2 -9609.089} C_VEL
LIN {X 0,Y 429.864,Z 471.66,A -85,B 0,C 180,E1 -9609.21,E2 -9609.21} C_VEL
LIN {X 0,Y 430.559,Z 416.771,A -85,B 0,C 180,E1 -9610.16,E2 -9610.16} C_VEL
LIN {X 0,Y 426.84,Z 397.325,A -85,B 0,C 180,E1 -9610.685,E2 -9610.685} C_VEL
LIN {X 0,Y 427.137,Z 388.324,A -85,B 0,C 180,E1 -9612.771,E2 -9612.771} C_VEL
LIN {X 0,Y 425.404,Z 378.497,A -85,B 0,C 180,E1 -9615.223,E2 -9615.223} C_VEL
LIN {X 0,Y 425.358,Z 378.504,A -85,B 0,C 180,E1 -9618.563,E2 -9618.563} C_VEL
LIN {X 0,Y 425.442,Z 378.486,A -85,B 0,C 180,E1 -9621.449,E2 -9621.449} C_VEL
LIN {X 0,Y 425.545,Z 378.479,A -85,B 0,C 180,E1 -9624.312,E2 -9624.312} C_VEL
LIN {X 0,Y 425.578,Z 378.473,A -85,B 0,C 180,E1 -9628.106,E2 -9628.106} C_VEL
LIN {X 0,Y 425.706,Z 378.456,A -85,B 0,C 180,E1 -9629.999,E2 -9629.999} C_VEL
LIN {X 0,Y 425.56,Z 378.473,A -85,B 0,C 180,E1 -9632.839,E2 -9632.839} C_VEL
LIN {X 0,Y 425.534,Z 378.477,A -85,B 0,C 180,E1 -9636.638,E2 -9636.638} C_VEL
LIN {X 0,Y 425.402,Z 378.492,A -85,B 0,C 180,E1 -9639.508,E2 -9639.508} C_VEL
LIN {X 0,Y 425.395,Z 378.492,A -85,B 0,C 180,E1 -9642.902,E2 -9642.902} C_VEL
LIN {X 0,Y 425.371,Z 378.496,A -85,B 0,C 180,E1 -9646.608,E2 -9646.608} C_VEL
LIN {X 0,Y 425.329,Z 378.504,A -85,B 0,C 180,E1 -9649.634,E2 -9649.634} C_VEL
LIN {X 0,Y 425.287,Z 378.508,A -85,B 0,C 180,E1 -9652.337,E2 -9652.337} C_VEL
LIN {X 0,Y 425.289,Z 378.508,A -85,B 0,C 180,E1 -9655.444,E2 -9655.444} C_VEL
LIN {X 0,Y 425.336,Z 378.499,A -85,B 0,C 180,E1 -9658.63,E2 -9658.63} C_VEL
LIN {X 0,Y 425.271,Z 378.512,A -85,B 0,C 180,E1 -9661.925,E2 -9661.925} C_VEL
LIN {X 0,Y 425.297,Z 378.508,A -85,B 0,C 180,E1 -9665.334,E2 -9665.334} C_VEL
LIN {X 0,Y 425.308,Z 378.504,A -85,B 0,C 180,E1 -9669.045,E2 -9669.045} C_VEL
LIN {X 0,Y 425.311,Z 378.505,A -85,B 0,C 180,E1 -9671.961,E2 -9671.961} C_VEL
LIN {X 0,Y 425.348,Z 378.605,A -85,B 0,C 180,E1 -9675.865,E2 -9675.865} C_VEL
LIN {X 0,Y 426.756,Z 386.419,A -85,B 0,C 180,E1 -9677.529,E2 -9677.529} C_VEL
LIN {X 0,Y 426.581,Z 396.319,A -85,B 0,C 180,E1 -9679.531,E2 -9679.531} C_VEL
LIN {X 0,Y 430.234,Z 416.326,A -85,B 0,C 180,E1 -9680.065,E2 -9680.065} C_VEL
LIN {X 0,Y 428.945,Z 504.745,A -85,B 0,C 180,E1 -9681.713,E2 -9681.713} C_VEL
LIN {X 0,Y 428.577,Z 517.692,A -85,B 0,C 180,E1 -9682.131,E2 -9682.131} C_VEL
LIN {X 0,Y 428.098,Z 530.706,A -85,B 0,C 180,E1 -9682.759,E2 -9682.759} C_VEL
LIN {X 0,Y 427.577,Z 542.004,A -85,B 0,C 180,E1 -9683.483,E2 -9683.483} C_VEL
LIN {X 0,Y 426.977,Z 553.106,A -85,B 0,C 180,E1 -9684.389,E2 -9684.389} C_VEL
LIN {X 0,Y 426.332,Z 563.979,A -85,B 0,C 180,E1 -9685.509,E2 -9685.509} C_VEL
LIN {X 0,Y 425.769,Z 573.466,A -85,B 0,C 180,E1 -9686.712,E2 -9686.712} C_VEL
LIN {X 0,Y 425.28,Z 582.106,A -85,B 0,C 180,E1 -9688.074,E2 -9688.074} C_VEL
LIN {X 0,Y 424.793,Z 589.665,A -85,B 0,C 180,E1 -9689.552,E2 -9689.552} C_VEL
LIN {X 0,Y 424.562,Z 594.678,A -85,B 0,C 180,E1 -9690.769,E2 -9690.769} C_VEL
LIN {X 0,Y 424.306,Z 599.923,A -85,B 0,C 180,E1 -9692.369,E2 -9692.369} C_VEL
LIN {X 0,Y 424.149,Z 603.732,A -85,B 0,C 180,E1 -9693.974,E2 -9693.974} C_VEL
LIN {X 0,Y 424.006,Z 606.455,A -85,B 0,C 180,E1 -9695.728,E2 -9695.728} C_VEL
LIN {X 0,Y 423.951,Z 607.247,A -85,B 0,C 180,E1 -9696.555,E2 -9696.555} C_VEL
LIN {X 0,Y 423.932,Z 607.881,A -85,B 0,C 180,E1 -9698.178,E2 -9698.178} C_VEL
LIN {X 0,Y 424.003,Z 607.416,A -85,B 0,C 180,E1 -9699.63,E2 -9699.63} C_VEL
LIN {X 0,Y 424.04,Z 606.252,A -85,B 0,C 180,E1 -9700.853,E2 -9700.853} C_VEL
LIN {X 0,Y 424.202,Z 603.311,A -85,B 0,C 180,E1 -9702.649,E2 -9702.649} C_VEL
LIN {X 0,Y 424.392,Z 599.324,A -85,B 0,C 180,E1 -9704.243,E2 -9704.243} C_VEL
LIN {X 0,Y 424.689,Z 594.727,A -85,B 0,C 180,E1 -9705.627,E2 -9705.627} C_VEL
LIN {X 0,Y 425.144,Z 587.904,A -85,B 0,C 180,E1 -9707.237,E2 -9707.237} C_VEL
LIN {X 0,Y 425.616,Z 580.77,A -85,B 0,C 180,E1 -9708.571,E2 -9708.571} C_VEL
LIN {X 0,Y 426.26,Z 571.06,A -85,B 0,C 180,E1 -9710.031,E2 -9710.031} C_VEL
LIN {X 0,Y 426.97,Z 560.828,A -85,B 0,C 180,E1 -9711.255,E2 -9711.255} C_VEL
LIN {X 0,Y 427.743,Z 549.574,A -85,B 0,C 180,E1 -9712.328,E2 -9712.328} C_VEL
LIN {X 0,Y 428.355,Z 538.502,A -85,B 0,C 180,E1 -9713.168,E2 -9713.168} C_VEL
LIN {X 0,Y 428.904,Z 526.158,A -85,B 0,C 180,E1 -9713.886,E2 -9713.886} C_VEL
LIN {X 0,Y 429.344,Z 512.75,A -85,B 0,C 180,E1 -9714.452,E2 -9714.452} C_VEL
LIN {X 0,Y 429.682,Z 499.077,A -85,B 0,C 180,E1 -9714.809,E2 -9714.809} C_VEL
LIN {X 0,Y 431.086,Z 416.567,A -85,B 0,C 180,E1 -9716.39,E2 -9716.39} C_VEL
LIN {X 0,Y 427.517,Z 399.032,A -85,B 0,C 180,E1 -9716.948,E2 -9716.948} C_VEL
LIN {X 0,Y 427.055,Z 396.935,A -85,B 0,C 180,E1 -9717.037,E2 -9717.037} C_VEL
LIN {X 0,Y 427.242,Z 387.961,A -85,B 0,C 180,E1 -9718.822,E2 -9718.822} C_VEL
LIN {X 0,Y 425.938,Z 380.011,A -85,B 0,C 180,E1 -9720.473,E2 -9720.473} C_VEL
LIN {X 0,Y 425.56,Z 378.478,A -85,B 0,C 180,E1 -9720.828,E2 -9720.828} C_VEL
LIN {X 0,Y 425.548,Z 378.481,A -85,B 0,C 180,E1 -9722.84,E2 -9722.84} C_VEL
LIN {X 0,Y 425.52,Z 378.482,A -85,B 0,C 180,E1 -9726.639,E2 -9726.639} C_VEL
LIN {X 0,Y 425.393,Z 378.496,A -85,B 0,C 180,E1 -9729.509,E2 -9729.509} C_VEL
LIN {X 0,Y 425.393,Z 378.496,A -85,B 0,C 180,E1 -9732.911,E2 -9732.911} C_VEL
LIN {X 0,Y 425.359,Z 378.501,A -85,B 0,C 180,E1 -9736.609,E2 -9736.609} C_VEL
LIN {X 0,Y 425.352,Z 378.503,A -85,B 0,C 180,E1 -9739.649,E2 -9739.649} C_VEL
LIN {X 0,Y 425.327,Z 378.504,A -85,B 0,C 180,E1 -9742.337,E2 -9742.337} C_VEL
LIN {X 0,Y 425.292,Z 378.509,A -85,B 0,C 180,E1 -9745.446,E2 -9745.446} C_VEL
LIN {X 0,Y 425.328,Z 378.503,A -85,B 0,C 180,E1 -9748.632,E2 -9748.632} C_VEL
LIN {X 0,Y 425.265,Z 378.514,A -85,B 0,C 180,E1 -9751.927,E2 -9751.927} C_VEL
LIN {X 0,Y 425.292,Z 378.51,A -85,B 0,C 180,E1 -9755.337,E2 -9755.337} C_VEL
LIN {X 0,Y 425.295,Z 378.509,A -85,B 0,C 180,E1 -9759.046,E2 -9759.046} C_VEL
LIN {X 0,Y 425.271,Z 378.51,A -85,B 0,C 180,E1 -9762.654,E2 -9762.654} C_VEL
LIN {X 0,Y 425.262,Z 378.509,A -85,B 0,C 180,E1 -9766.046,E2 -9766.046} C_VEL
LIN {X 0,Y 425.269,Z 378.511,A -85,B 0,C 180,E1 -9768.623,E2 -9768.623} C_VEL
LIN {X 0,Y 425.307,Z 378.508,A -85,B 0,C 180,E1 -9771.104,E2 -9771.104} C_VEL
LIN {X 0,Y 425.296,Z 378.51,A -85,B 0,C 180,E1 -9774.666,E2 -9774.666} C_VEL
LIN {X 0,Y 425.271,Z 378.51,A -85,B 0,C 180,E1 -9778.075,E2 -9778.075} C_VEL
LIN {X 0,Y 425.335,Z 378.504,A -85,B 0,C 180,E1 -9781.37,E2 -9781.37} C_VEL
LIN {X 0,Y 425.412,Z 378.614,A -85,B 0,C 180,E1 -9782.912,E2 -9782.912} C_VEL
LIN {X 0,Y 427.924,Z 391.684,A -85,B 0,C 180,E1 -9785.76,E2 -9785.76} C_VEL
LIN {X 0,Y 428.121,Z 395.477,A -85,B 0,C 180,E1 -9786.543,E2 -9786.543} C_VEL
LIN {X 0,Y 427.012,Z 413.101,A -85,B 0,C 180,E1 -9790.032,E2 -9790.032} C_VEL
LIN {X 0,Y 426.65,Z 419.625,A -85,B 0,C 180,E1 -9791.298,E2 -9791.298} C_VEL
LIN {X 0,Y 430.246,Z 442.868,A -85,B 0,C 180,E1 -9791.912,E2 -9791.912} C_VEL
LIN {X 0,Y 429.365,Z 528.293,A -85,B 0,C 180,E1 -9793.417,E2 -9793.417} C_VEL
LIN {X 0,Y 428.831,Z 542.081,A -85,B 0,C 180,E1 -9793.855,E2 -9793.855} C_VEL
LIN {X 0,Y 428.266,Z 555.027,A -85,B 0,C 180,E1 -9794.474,E2 -9794.474} C_VEL
LIN {X 0,Y 427.594,Z 566.818,A -85,B 0,C 180,E1 -9795.242,E2 -9795.242} C_VEL
LIN {X 0,Y 426.94,Z 577.229,A -85,B 0,C 180,E1 -9796.102,E2 -9796.102} C_VEL
LIN {X 0,Y 426.281,Z 588.462,A -85,B 0,C 180,E1 -9797.262,E2 -9797.262} C_VEL
LIN {X 0,Y 425.607,Z 598.503,A -85,B 0,C 180,E1 -9798.572,E2 -9798.572} C_VEL
LIN {X 0,Y 425.045,Z 607.346,A -85,B 0,C 180,E1 -9800.003,E2 -9800.003} C_VEL
LIN {X 0,Y 424.638,Z 614.399,A -85,B 0,C 180,E1 -9801.435,E2 -9801.435} C_VEL
LIN {X 0,Y 424.355,Z 620.037,A -85,B 0,C 180,E1 -9802.866,E2 -9802.866} C_VEL
LIN {X 0,Y 424.192,Z 624.463,A -85,B 0,C 180,E1 -9804.296,E2 -9804.296} C_VEL
LIN {X 0,Y 424.2,Z 626.801,A -85,B 0,C 180,E1 -9805.25,E2 -9805.25} C_VEL
LIN {X 0,Y 424.098,Z 628.701,A -85,B 0,C 180,E1 -9806.201,E2 -9806.201} C_VEL
LIN {X 0,Y 424.131,Z 630.142,A -85,B 0,C 180,E1 -9807.152,E2 -9807.152} C_VEL
LIN {X 0,Y 424.128,Z 631.158,A -85,B 0,C 180,E1 -9808.102,E2 -9808.102} C_VEL
LIN {X 0,Y 424.084,Z 632.012,A -85,B 0,C 180,E1 -9810.001,E2 -9810.001} C_VEL
LIN {X 0,Y 424.088,Z 631.81,A -85,B 0,C 180,E1 -9810.951,E2 -9810.951} C_VEL
LIN {X 0,Y 424.129,Z 631.202,A -85,B 0,C 180,E1 -9811.9,E2 -9811.9} C_VEL
LIN {X 0,Y 424.131,Z 630.201,A -85,B 0,C 180,E1 -9812.851,E2 -9812.851} C_VEL
LIN {X 0,Y 424.099,Z 628.797,A -85,B 0,C 180,E1 -9813.802,E2 -9813.802} C_VEL
LIN {X 0,Y 424.21,Z 625.843,A -85,B 0,C 180,E1 -9815.229,E2 -9815.229} C_VEL
LIN {X 0,Y 424.302,Z 621.844,A -85,B 0,C 180,E1 -9816.659,E2 -9816.659} C_VEL
LIN {X 0,Y 424.585,Z 615.701,A -85,B 0,C 180,E1 -9818.329,E2 -9818.329} C_VEL
LIN {X 0,Y 424.964,Z 608.983,A -85,B 0,C 180,E1 -9819.761,E2 -9819.761} C_VEL
LIN {X 0,Y 425.485,Z 600.65,A -85,B 0,C 180,E1 -9821.192,E2 -9821.192} C_VEL
LIN {X 0,Y 426.177,Z 592.118,A -85,B 0,C 180,E1 -9822.38,E2 -9822.38} C_VEL
LIN {X 0,Y 426.759,Z 582.129,A -85,B 0,C 180,E1 -9823.517,E2 -9823.517} C_VEL
LIN {X 0,Y 427.457,Z 571.159,A -85,B 0,C 180,E1 -9824.522,E2 -9824.522} C_VEL
LIN {X 0,Y 428.172,Z 559.752,A -85,B 0,C 180,E1 -9825.349,E2 -9825.349} C_VEL
LIN {X 0,Y 428.821,Z 548.065,A -85,B 0,C 180,E1 -9825.995,E2 -9825.995} C_VEL
LIN {X 0,Y 429.329,Z 535.59,A -85,B 0,C 180,E1 -9826.495,E2 -9826.495} C_VEL
LIN {X 0,Y 429.797,Z 523.092,A -85,B 0,C 180,E1 -9826.813,E2 -9826.813} C_VEL
LIN {X 0,Y 430.622,Z 443.343,A -85,B 0,C 180,E1 -9828.213,E2 -9828.213} C_VEL
LIN {X 0,Y 426.704,Z 419.12,A -85,B 0,C 180,E1 -9828.861,E2 -9828.861} C_VEL
LIN {X 0,Y 427.897,Z 401.106,A -85,B 0,C 180,E1 -9832.442,E2 -9832.442} C_VEL
LIN {X 0,Y 428.313,Z 393.61,A -85,B 0,C 180,E1 -9833.962,E2 -9833.962} C_VEL
LIN {X 0,Y 426.208,Z 382.449,A -85,B 0,C 180,E1 -9836.438,E2 -9836.438} C_VEL
LIN {X 0,Y 425.358,Z 378.504,A -85,B 0,C 180,E1 -9837.369,E2 -9837.369} C_VEL
LIN {X 0,Y 425.293,Z 378.51,A -85,B 0,C 180,E1 -9840.817,E2 -9840.817} C_VEL
LIN {X 0,Y 425.317,Z 378.504,A -85,B 0,C 180,E1 -9844.289,E2 -9844.289} C_VEL
LIN {X 0,Y 425.285,Z 378.512,A -85,B 0,C 180,E1 -9847.695,E2 -9847.695} C_VEL
LIN {X 0,Y 425.287,Z 378.512,A -85,B 0,C 180,E1 -9850.521,E2 -9850.521} C_VEL
LIN {X 0,Y 425.263,Z 378.516,A -85,B 0,C 180,E1 -9853.351,E2 -9853.351} C_VEL
LIN {X 0,Y 425.264,Z 378.515,A -85,B 0,C 180,E1 -9856.65,E2 -9856.65} C_VEL
LIN {X 0,Y 425.291,Z 378.503,A -85,B 0,C 180,E1 -9859.873,E2 -9859.873} C_VEL
LIN {X 0,Y 425.283,Z 378.51,A -85,B 0,C 180,E1 -9862.489,E2 -9862.489} C_VEL
LIN {X 0,Y 425.313,Z 378.5,A -85,B 0,C 180,E1 -9865.818,E2 -9865.818} C_VEL
LIN {X 0,Y 425.296,Z 378.501,A -85,B 0,C 180,E1 -9869.239,E2 -9869.239} C_VEL
LIN {X 0,Y 425.354,Z 378.502,A -85,B 0,C 180,E1 -9872.443,E2 -9872.443} C_VEL
LIN {X 0,Y 425.353,Z 378.498,A -85,B 0,C 180,E1 -9875.602,E2 -9875.602} C_VEL
LIN {X 0,Y 425.299,Z 378.51,A -85,B 0,C 180,E1 -9878.682,E2 -9878.682} C_VEL
LIN {X 0,Y 425.338,Z 378.495,A -85,B 0,C 180,E1 -9881.703,E2 -9881.703} C_VEL
LIN {X 0,Y 425.354,Z 378.496,A -85,B 0,C 180,E1 -9884.671,E2 -9884.671} C_VEL
LIN {X 0,Y 425.418,Z 378.491,A -85,B 0,C 180,E1 -9887.598,E2 -9887.598} C_VEL
LIN {X 0,Y 425.449,Z 378.487,A -85,B 0,C 180,E1 -9891.45,E2 -9891.45} C_VEL
LIN {X 0,Y 425.56,Z 378.475,A -85,B 0,C 180,E1 -9894.313,E2 -9894.313} C_VEL
LIN {X 0,Y 425.579,Z 378.473,A -85,B 0,C 180,E1 -9898.107,E2 -9898.107} C_VEL
LIN {X 0,Y 425.707,Z 378.457,A -85,B 0,C 180,E1 -9900,E2 -9900} C_VEL
LIN {X 0,Y 425.552,Z 378.473,A -85,B 0,C 180,E1 -9902.84,E2 -9902.84} C_VEL
LIN {X 0,Y 425.537,Z 378.474,A -85,B 0,C 180,E1 -9906.639,E2 -9906.639} C_VEL
LIN {X 0,Y 425.407,Z 378.494,A -85,B 0,C 180,E1 -9909.509,E2 -9909.509} C_VEL
LIN {X 0,Y 425.4,Z 378.494,A -85,B 0,C 180,E1 -9912.904,E2 -9912.904} C_VEL
LIN {X 0,Y 425.368,Z 378.498,A -85,B 0,C 180,E1 -9916.605,E2 -9916.605} C_VEL
LIN {X 0,Y 425.335,Z 378.506,A -85,B 0,C 180,E1 -9919.636,E2 -9919.636} C_VEL
LIN {X 0,Y 425.311,Z 378.507,A -85,B 0,C 180,E1 -9923.365,E2 -9923.365} C_VEL
LIN {X 0,Y 425.353,Z 378.503,A -85,B 0,C 180,E1 -9926.844,E2 -9926.844} C_VEL
LIN {X 0,Y 425.373,Z 378.543,A -85,B 0,C 180,E1 -9928.427,E2 -9928.427} C_VEL
LIN {X 0,Y 427.32,Z 388.864,A -85,B 0,C 180,E1 -9931.074,E2 -9931.074} C_VEL
LIN {X 0,Y 427.243,Z 395.247,A -85,B 0,C 180,E1 -9932.597,E2 -9932.597} C_VEL
LIN {X 0,Y 427.095,Z 397.96,A -85,B 0,C 180,E1 -9933.232,E2 -9933.232} C_VEL
LIN {X 0,Y 430.954,Z 417.179,A -85,B 0,C 180,E1 -9933.78,E2 -9933.78} C_VEL
LIN {X 0,Y 429.733,Z 505.163,A -85,B 0,C 180,E1 -9935.338,E2 -9935.338} C_VEL
LIN {X 0,Y 429.341,Z 518.813,A -85,B 0,C 180,E1 -9935.78,E2 -9935.78} C_VEL
LIN {X 0,Y 428.844,Z 531.567,A -85,B 0,C 180,E1 -9936.396,E2 -9936.396} C_VEL
LIN {X 0,Y 428.281,Z 541.849,A -85,B 0,C 180,E1 -9937.054,E2 -9937.054} C_VEL
LIN {X 0,Y 427.576,Z 553.615,A -85,B 0,C 180,E1 -9938.021,E2 -9938.021} C_VEL
LIN {X 0,Y 426.927,Z 563.135,A -85,B 0,C 180,E1 -9938.992,E2 -9938.992} C_VEL
LIN {X 0,Y 426.201,Z 572.605,A -85,B 0,C 180,E1 -9940.172,E2 -9940.172} C_VEL
LIN {X 0,Y 425.675,Z 580.217,A -85,B 0,C 180,E1 -9941.332,E2 -9941.332} C_VEL
LIN {X 0,Y 425.187,Z 587.416,A -85,B 0,C 180,E1 -9942.664,E2 -9942.664} C_VEL
LIN {X 0,Y 424.822,Z 593.33,A -85,B 0,C 180,E1 -9944.013,E2 -9944.013} C_VEL
LIN {X 0,Y 424.491,Z 598.19,A -85,B 0,C 180,E1 -9945.392,E2 -9945.392} C_VEL
LIN {X 0,Y 424.224,Z 602.985,A -85,B 0,C 180,E1 -9947.215,E2 -9947.215} C_VEL
LIN {X 0,Y 424.118,Z 605.346,A -85,B 0,C 180,E1 -9948.482,E2 -9948.482} C_VEL
LIN {X 0,Y 423.983,Z 606.956,A -85,B 0,C 180,E1 -9949.723,E2 -9949.723} C_VEL
LIN {X 0,Y 423.933,Z 607.935,A -85,B 0,C 180,E1 -9951.185,E2 -9951.185} C_VEL
LIN {X 0,Y 423.951,Z 607.945,A -85,B 0,C 180,E1 -9952.723,E2 -9952.723} C_VEL
LIN {X 0,Y 424.018,Z 606.585,A -85,B 0,C 180,E1 -9954.54,E2 -9954.54} C_VEL
LIN {X 0,Y 424.121,Z 604.525,A -85,B 0,C 180,E1 -9955.949,E2 -9955.949} C_VEL
LIN {X 0,Y 424.359,Z 600.797,A -85,B 0,C 180,E1 -9957.633,E2 -9957.633} C_VEL
LIN {X 0,Y 424.581,Z 596.267,A -85,B 0,C 180,E1 -9959.126,E2 -9959.126} C_VEL
LIN {X 0,Y 424.966,Z 589.821,A -85,B 0,C 180,E1 -9960.758,E2 -9960.758} C_VEL
LIN {X 0,Y 425.448,Z 582.639,A -85,B 0,C 180,E1 -9962.181,E2 -9962.181} C_VEL
LIN {X 0,Y 425.983,Z 574.114,A -85,B 0,C 180,E1 -9963.546,E2 -9963.546} C_VEL
LIN {X 0,Y 426.647,Z 564.202,A -85,B 0,C 180,E1 -9964.828,E2 -9964.828} C_VEL
LIN {X 0,Y 427.41,Z 552.885,A -85,B 0,C 180,E1 -9965.984,E2 -9965.984} C_VEL
LIN {X 0,Y 427.982,Z 542.088,A -85,B 0,C 180,E1 -9966.867,E2 -9966.867} C_VEL
LIN {X 0,Y 428.579,Z 529.685,A -85,B 0,C 180,E1 -9967.651,E2 -9967.651} C_VEL
LIN {X 0,Y 429.105,Z 516.233,A -85,B 0,C 180,E1 -9968.265,E2 -9968.265} C_VEL
LIN {X 0,Y 429.493,Z 503.169,A -85,B 0,C 180,E1 -9968.656,E2 -9968.656} C_VEL
LIN {X 0,Y 429.864,Z 471.66,A -85,B 0,C 180,E1 -9969.21,E2 -9969.21} C_VEL
LIN {X 0,Y 429.319,Z 465.852,A -85,B 0,C 180,E1 -9969.335,E2 -9969.335} C_VEL
LIN {X 0,Y 424.009,Z 447.173,A -85,B 0,C 180,E1 -9969.884,E2 -9969.884} C_VEL
LIN {X 0,Y 423.484,Z 441.365,A -85,B 0,C 180,E1 -9970.011,E2 -9970.011} C_VEL
LIN {X 0,Y 423.732,Z 417.458,A -85,B 0,C 180,E1 -9970.437,E2 -9970.437} C_VEL
LIN {X 0,Y 419.885,Z 397.539,A -85,B 0,C 180,E1 -9970.981,E2 -9970.981} C_VEL
LIN {X 0,Y 420.224,Z 390.073,A -85,B 0,C 180,E1 -9972.73,E2 -9972.73} C_VEL
LIN {X 0,Y 418.35,Z 379.375,A -85,B 0,C 180,E1 -9975.435,E2 -9975.435} C_VEL
LIN {X 0,Y 418.321,Z 379.378,A -85,B 0,C 180,E1 -9978.368,E2 -9978.368} C_VEL
LIN {X 0,Y 418.402,Z 379.363,A -85,B 0,C 180,E1 -9981.304,E2 -9981.304} C_VEL
LIN {X 0,Y 418.503,Z 379.355,A -85,B 0,C 180,E1 -9984.216,E2 -9984.216} C_VEL
LIN {X 0,Y 418.547,Z 379.349,A -85,B 0,C 180,E1 -9988.074,E2 -9988.074} C_VEL
LIN {X 0,Y 418.675,Z 379.332,A -85,B 0,C 180,E1 -9989.999,E2 -9989.999} C_VEL
LIN {X 0,Y 418.513,Z 379.35,A -85,B 0,C 180,E1 -9992.886,E2 -9992.886} C_VEL
LIN {X 0,Y 418.497,Z 379.353,A -85,B 0,C 180,E1 -9996.75,E2 -9996.75} C_VEL
LIN {X 0,Y 418.402,Z 379.365,A -85,B 0,C 180,E1 -9998.694,E2 -9998.694} C_VEL
LIN {X 0,Y 418.357,Z 379.37,A -85,B 0,C 180,E1 -10002.613,E2 -10002.613} C_VEL
LIN {X 0,Y 418.312,Z 379.376,A -85,B 0,C 180,E1 -10005.592,E2 -10005.592} C_VEL
LIN {X 0,Y 418.284,Z 379.379,A -85,B 0,C 180,E1 -10008.615,E2 -10008.615} C_VEL
LIN {X 0,Y 418.234,Z 379.388,A -85,B 0,C 180,E1 -10011.695,E2 -10011.695} C_VEL
LIN {X 0,Y 418.282,Z 379.378,A -85,B 0,C 180,E1 -10014.863,E2 -10014.863} C_VEL
LIN {X 0,Y 418.293,Z 379.381,A -85,B 0,C 180,E1 -10018.062,E2 -10018.062} C_VEL
LIN {X 0,Y 418.22,Z 379.389,A -85,B 0,C 180,E1 -10021.394,E2 -10021.394} C_VEL
LIN {X 0,Y 418.262,Z 379.38,A -85,B 0,C 180,E1 -10024.579,E2 -10024.579} C_VEL
LIN {X 0,Y 418.234,Z 379.388,A -85,B 0,C 180,E1 -10027.834,E2 -10027.834} C_VEL
LIN {X 0,Y 418.26,Z 379.382,A -85,B 0,C 180,E1 -10030.941,E2 -10030.941} C_VEL
LIN {X 0,Y 418.211,Z 379.393,A -85,B 0,C 180,E1 -10033.729,E2 -10033.729} C_VEL
LIN {X 0,Y 418.32,Z 379.515,A -85,B 0,C 180,E1 -10035.711,E2 -10035.711} C_VEL
LIN {X 0,Y 419.782,Z 387.57,A -85,B 0,C 180,E1 -10037.444,E2 -10037.444} C_VEL
LIN {X 0,Y 419.611,Z 396.346,A -85,B 0,C 180,E1 -10039.238,E2 -10039.238} C_VEL
LIN {X 0,Y 423.419,Z 417.09,A -85,B 0,C 180,E1 -10039.814,E2 -10039.814} C_VEL
LIN {X 0,Y 422.063,Z 505.396,A -85,B 0,C 180,E1 -10041.499,E2 -10041.499} C_VEL
LIN {X 0,Y 421.661,Z 518.197,A -85,B 0,C 180,E1 -10041.925,E2 -10041.925} C_VEL
LIN {X 0,Y 421.177,Z 530.951,A -85,B 0,C 180,E1 -10042.553,E2 -10042.553} C_VEL
LIN {X 0,Y 420.601,Z 542.719,A -85,B 0,C 180,E1 -10043.324,E2 -10043.324} C_VEL
LIN {X 0,Y 419.96,Z 554.335,A -85,B 0,C 180,E1 -10044.308,E2 -10044.308} C_VEL
LIN {X 0,Y 419.325,Z 564.701,A -85,B 0,C 180,E1 -10045.406,E2 -10045.406} C_VEL
LIN {X 0,Y 418.756,Z 573.732,A -85,B 0,C 180,E1 -10046.578,E2 -10046.578} C_VEL
LIN {X 0,Y 418.218,Z 582.785,A -85,B 0,C 180,E1 -10048.038,E2 -10048.038} C_VEL
LIN {X 0,Y 417.777,Z 589.491,A -85,B 0,C 180,E1 -10049.373,E2 -10049.373} C_VEL
LIN {X 0,Y 417.466,Z 595.202,A -85,B 0,C 180,E1 -10050.777,E2 -10050.777} C_VEL
LIN {X 0,Y 417.216,Z 600.353,A -85,B 0,C 180,E1 -10052.404,E2 -10052.404} C_VEL
LIN {X 0,Y 417.063,Z 604.055,A -85,B 0,C 180,E1 -10054.015,E2 -10054.015} C_VEL
LIN {X 0,Y 416.931,Z 606.421,A -85,B 0,C 180,E1 -10055.536,E2 -10055.536} C_VEL
LIN {X 0,Y 416.816,Z 607.803,A -85,B 0,C 180,E1 -10057.182,E2 -10057.182} C_VEL
LIN {X 0,Y 416.86,Z 608.071,A -85,B 0,C 180,E1 -10058.228,E2 -10058.228} C_VEL
LIN {X 0,Y 416.87,Z 607.815,A -85,B 0,C 180,E1 -10059.265,E2 -10059.265} C_VEL
LIN {X 0,Y 416.945,Z 606.685,A -85,B 0,C 180,E1 -10060.718,E2 -10060.718} C_VEL
LIN {X 0,Y 417.097,Z 604.289,A -85,B 0,C 180,E1 -10062.344,E2 -10062.344} C_VEL
LIN {X 0,Y 417.259,Z 601.22,A -85,B 0,C 180,E1 -10063.747,E2 -10063.747} C_VEL
LIN {X 0,Y 417.547,Z 596.395,A -85,B 0,C 180,E1 -10065.376,E2 -10065.376} C_VEL
LIN {X 0,Y 417.948,Z 590.711,A -85,B 0,C 180,E1 -10066.846,E2 -10066.846} C_VEL
LIN {X 0,Y 418.482,Z 583.222,A -85,B 0,C 180,E1 -10068.374,E2 -10068.374} C_VEL
LIN {X 0,Y 419.154,Z 574.102,A -85,B 0,C 180,E1 -10069.86,E2 -10069.86} C_VEL
LIN {X 0,Y 419.892,Z 563.648,A -85,B 0,C 180,E1 -10071.206,E2 -10071.206} C_VEL
LIN {X 0,Y 420.655,Z 552.846,A -85,B 0,C 180,E1 -10072.319,E2 -10072.319} C_VEL
LIN {X 0,Y 421.403,Z 540.763,A -85,B 0,C 180,E1 -10073.296,E2 -10073.296} C_VEL
LIN {X 0,Y 422.059,Z 528.037,A -85,B 0,C 180,E1 -10074.086,E2 -10074.086} C_VEL
LIN {X 0,Y 422.558,Z 514.512,A -85,B 0,C 180,E1 -10074.692,E2 -10074.692} C_VEL
LIN {X 0,Y 422.911,Z 502.199,A -85,B 0,C 180,E1 -10075.054,E2 -10075.054} C_VEL
LIN {X 0,Y 424.456,Z 417.535,A -85,B 0,C 180,E1 -10076.721,E2 -10076.721} C_VEL
LIN {X 0,Y 421.082,Z 400.946,A -85,B 0,C 180,E1 -10077.264,E2 -10077.264} C_VEL
LIN {X 0,Y 420.251,Z 397.074,A -85,B 0,C 180,E1 -10077.424,E2 -10077.424} C_VEL
LIN {X 0,Y 420.343,Z 389.057,A -85,B 0,C 180,E1 -10079.042,E2 -10079.042} C_VEL
LIN {X 0,Y 418.93,Z 381.145,A -85,B 0,C 180,E1 -10080.721,E2 -10080.721} C_VEL
LIN {X 0,Y 418.506,Z 379.357,A -85,B 0,C 180,E1 -10081.143,E2 -10081.143} C_VEL
LIN {X 0,Y 418.502,Z 379.359,A -85,B 0,C 180,E1 -10082.888,E2 -10082.888} C_VEL
LIN {X 0,Y 418.483,Z 379.359,A -85,B 0,C 180,E1 -10086.751,E2 -10086.751} C_VEL
LIN {X 0,Y 418.35,Z 379.374,A -85,B 0,C 180,E1 -10089.671,E2 -10089.671} C_VEL
LIN {X 0,Y 418.344,Z 379.374,A -85,B 0,C 180,E1 -10093.007,E2 -10093.007} C_VEL
LIN {X 0,Y 418.309,Z 379.378,A -85,B 0,C 180,E1 -10096.739,E2 -10096.739} C_VEL
LIN {X 0,Y 418.293,Z 379.382,A -85,B 0,C 180,E1 -10099.804,E2 -10099.804} C_VEL
LIN {X 0,Y 418.28,Z 379.379,A -85,B 0,C 180,E1 -10102.734,E2 -10102.734} C_VEL
LIN {X 0,Y 418.265,Z 379.385,A -85,B 0,C 180,E1 -10105.904,E2 -10105.904} C_VEL
LIN {X 0,Y 418.265,Z 379.384,A -85,B 0,C 180,E1 -10109.162,E2 -10109.162} C_VEL
LIN {X 0,Y 418.251,Z 379.384,A -85,B 0,C 180,E1 -10112.846,E2 -10112.846} C_VEL
LIN {X 0,Y 418.24,Z 379.386,A -85,B 0,C 180,E1 -10116.24,E2 -10116.24} C_VEL
LIN {X 0,Y 418.247,Z 379.388,A -85,B 0,C 180,E1 -10119.682,E2 -10119.682} C_VEL
LIN {X 0,Y 418.224,Z 379.387,A -85,B 0,C 180,E1 -10122.323,E2 -10122.323} C_VEL
LIN {X 0,Y 418.235,Z 379.39,A -85,B 0,C 180,E1 -10125.111,E2 -10125.111} C_VEL
LIN {X 0,Y 418.236,Z 379.386,A -85,B 0,C 180,E1 -10127.768,E2 -10127.768} C_VEL
LIN {X 0,Y 418.251,Z 379.386,A -85,B 0,C 180,E1 -10130.62,E2 -10130.62} C_VEL
LIN {X 0,Y 418.241,Z 379.385,A -85,B 0,C 180,E1 -10133.978,E2 -10133.978} C_VEL
LIN {X 0,Y 418.257,Z 379.387,A -85,B 0,C 180,E1 -10137.157,E2 -10137.157} C_VEL
LIN {X 0,Y 418.272,Z 379.385,A -85,B 0,C 180,E1 -10140.84,E2 -10140.84} C_VEL
LIN {X 0,Y 418.374,Z 379.555,A -85,B 0,C 180,E1 -10142.677,E2 -10142.677} C_VEL
LIN {X 0,Y 420.919,Z 392.68,A -85,B 0,C 180,E1 -10145.593,E2 -10145.593} C_VEL
LIN {X 0,Y 421.191,Z 396.481,A -85,B 0,C 180,E1 -10146.394,E2 -10146.394} C_VEL
LIN {X 0,Y 420.098,Z 412.684,A -85,B 0,C 180,E1 -10149.662,E2 -10149.662} C_VEL
LIN {X 0,Y 419.716,Z 418.941,A -85,B 0,C 180,E1 -10150.901,E2 -10150.901} C_VEL
LIN {X 0,Y 423.503,Z 443.957,A -85,B 0,C 180,E1 -10151.651,E2 -10151.651} C_VEL
LIN {X 0,Y 422.534,Z 528.534,A -85,B 0,C 180,E1 -10153.172,E2 -10153.172} C_VEL
LIN {X 0,Y 421.959,Z 542.169,A -85,B 0,C 180,E1 -10153.616,E2 -10153.616} C_VEL
LIN {X 0,Y 421.439,Z 554.515,A -85,B 0,C 180,E1 -10154.216,E2 -10154.216} C_VEL
LIN {X 0,Y 420.713,Z 566.373,A -85,B 0,C 180,E1 -10154.995,E2 -10154.995} C_VEL
LIN {X 0,Y 419.958,Z 577.798,A -85,B 0,C 180,E1 -10155.958,E2 -10155.958} C_VEL
LIN {X 0,Y 419.291,Z 588.106,A -85,B 0,C 180,E1 -10157.046,E2 -10157.046} C_VEL
LIN {X 0,Y 418.749,Z 596.539,A -85,B 0,C 180,E1 -10158.137,E2 -10158.137} C_VEL
LIN {X 0,Y 418.071,Z 605.679,A -85,B 0,C 180,E1 -10159.59,E2 -10159.59} C_VEL
LIN {X 0,Y 417.651,Z 613.046,A -85,B 0,C 180,E1 -10161.047,E2 -10161.047} C_VEL
LIN {X 0,Y 417.365,Z 618.029,A -85,B 0,C 180,E1 -10162.259,E2 -10162.259} C_VEL
LIN {X 0,Y 417.167,Z 622.843,A -85,B 0,C 180,E1 -10163.707,E2 -10163.707} C_VEL
LIN {X 0,Y 417.107,Z 626.566,A -85,B 0,C 180,E1 -10165.169,E2 -10165.169} C_VEL
LIN {X 0,Y 417.014,Z 628.473,A -85,B 0,C 180,E1 -10166.136,E2 -10166.136} C_VEL
LIN {X 0,Y 417.028,Z 629.924,A -85,B 0,C 180,E1 -10167.103,E2 -10167.103} C_VEL
LIN {X 0,Y 417.056,Z 630.947,A -85,B 0,C 180,E1 -10168.07,E2 -10168.07} C_VEL
LIN {X 0,Y 417.004,Z 631.81,A -85,B 0,C 180,E1 -10170.001,E2 -10170.001} C_VEL
LIN {X 0,Y 417.01,Z 631.615,A -85,B 0,C 180,E1 -10170.967,E2 -10170.967} C_VEL
LIN {X 0,Y 417.056,Z 631.011,A -85,B 0,C 180,E1 -10171.933,E2 -10171.933} C_VEL
LIN {X 0,Y 417.028,Z 630.011,A -85,B 0,C 180,E1 -10172.899,E2 -10172.899} C_VEL
LIN {X 0,Y 417.014,Z 628.612,A -85,B 0,C 180,E1 -10173.867,E2 -10173.867} C_VEL
LIN {X 0,Y 417.125,Z 625.663,A -85,B 0,C 180,E1 -10175.318,E2 -10175.318} C_VEL
LIN {X 0,Y 417.235,Z 621.669,A -85,B 0,C 180,E1 -10176.773,E2 -10176.773} C_VEL
LIN {X 0,Y 417.526,Z 615.534,A -85,B 0,C 180,E1 -10178.471,E2 -10178.471} C_VEL
LIN {X 0,Y 417.93,Z 608.821,A -85,B 0,C 180,E1 -10179.927,E2 -10179.927} C_VEL
LIN {X 0,Y 418.501,Z 600.499,A -85,B 0,C 180,E1 -10181.382,E2 -10181.382} C_VEL
LIN {X 0,Y 419.217,Z 591.99,A -85,B 0,C 180,E1 -10182.589,E2 -10182.589} C_VEL
LIN {X 0,Y 419.848,Z 581.709,A -85,B 0,C 180,E1 -10183.778,E2 -10183.778} C_VEL
LIN {X 0,Y 420.589,Z 571.104,A -85,B 0,C 180,E1 -10184.764,E2 -10184.764} C_VEL
LIN {X 0,Y 421.332,Z 559.751,A -85,B 0,C 180,E1 -10185.604,E2 -10185.604} C_VEL
LIN {X 0,Y 422.011,Z 548.161,A -85,B 0,C 180,E1 -10186.261,E2 -10186.261} C_VEL
LIN {X 0,Y 422.537,Z 535.817,A -85,B 0,C 180,E1 -10186.768,E2 -10186.768} C_VEL
LIN {X 0,Y 423.065,Z 522.143,A -85,B 0,C 180,E1 -10187.119,E2 -10187.119} C_VEL
LIN {X 0,Y 423.863,Z 443.871,A -85,B 0,C 180,E1 -10188.52,E2 -10188.52} C_VEL
LIN {X 0,Y 419.798,Z 419.006,A -85,B 0,C 180,E1 -10189.187,E2 -10189.187} C_VEL
LIN {X 0,Y 420.968,Z 402.247,A -85,B 0,C 180,E1 -10192.582,E2 -10192.582} C_VEL
LIN {X 0,Y 421.366,Z 394.801,A -85,B 0,C 180,E1 -10194.12,E2 -10194.12} C_VEL
LIN {X 0,Y 419.221,Z 383.679,A -85,B 0,C 180,E1 -10196.645,E2 -10196.645} C_VEL
LIN {X 0,Y 418.321,Z 379.381,A -85,B 0,C 180,E1 -10197.68,E2 -10197.68} C_VEL
LIN {X 0,Y 418.244,Z 379.39,A -85,B 0,C 180,E1 -10201.02,E2 -10201.02} C_VEL
LIN {X 0,Y 418.254,Z 379.386,A -85,B 0,C 180,E1 -10203.678,E2 -10203.678} C_VEL
LIN {X 0,Y 418.246,Z 379.391,A -85,B 0,C 180,E1 -10207.225,E2 -10207.225} C_VEL
LIN {X 0,Y 418.257,Z 379.387,A -85,B 0,C 180,E1 -10209.682,E2 -10209.682} C_VEL
LIN {X 0,Y 418.235,Z 379.389,A -85,B 0,C 180,E1 -10212.322,E2 -10212.322} C_VEL
LIN {X 0,Y 418.241,Z 379.389,A -85,B 0,C 180,E1 -10215.109,E2 -10215.109} C_VEL
LIN {X 0,Y 418.246,Z 379.384,A -85,B 0,C 180,E1 -10217.767,E2 -10217.767} C_VEL
LIN {X 0,Y 418.255,Z 379.383,A -85,B 0,C 180,E1 -10220.62,E2 -10220.62} C_VEL
LIN {X 0,Y 418.248,Z 379.383,A -85,B 0,C 180,E1 -10223.976,E2 -10223.976} C_VEL
LIN {X 0,Y 418.263,Z 379.384,A -85,B 0,C 180,E1 -10227.156,E2 -10227.156} C_VEL
LIN {X 0,Y 418.274,Z 379.384,A -85,B 0,C 180,E1 -10230.896,E2 -10230.896} C_VEL
LIN {X 0,Y 418.274,Z 379.377,A -85,B 0,C 180,E1 -10234.096,E2 -10234.096} C_VEL
LIN {X 0,Y 418.243,Z 379.379,A -85,B 0,C 180,E1 -10237.264,E2 -10237.264} C_VEL
LIN {X 0,Y 418.289,Z 379.381,A -85,B 0,C 180,E1 -10240.364,E2 -10240.364} C_VEL
LIN {X 0,Y 418.323,Z 379.374,A -85,B 0,C 180,E1 -10243.405,E2 -10243.405} C_VEL
LIN {X 0,Y 418.352,Z 379.371,A -85,B 0,C 180,E1 -10247,E2 -10247} C_VEL
LIN {X 0,Y 418.347,Z 379.372,A -85,B 0,C 180,E1 -10250.329,E2 -10250.329} C_VEL
LIN {X 0,Y 418.52,Z 379.352,A -85,B 0,C 180,E1 -10252.28,E2 -10252.28} C_VEL
LIN {X 0,Y 418.519,Z 379.351,A -85,B 0,C 180,E1 -10254.217,E2 -10254.217} C_VEL
LIN {X 0,Y 418.548,Z 379.348,A -85,B 0,C 180,E1 -10258.076,E2 -10258.076} C_VEL
LIN {X 0,Y 418.677,Z 379.332,A -85,B 0,C 180,E1 -10260,E2 -10260} C_VEL
LIN {X 0,Y 418.507,Z 379.351,A -85,B 0,C 180,E1 -10262.888,E2 -10262.888} C_VEL
LIN {X 0,Y 418.5,Z 379.35,A -85,B 0,C 180,E1 -10266.751,E2 -10266.751} C_VEL
LIN {X 0,Y 418.407,Z 379.365,A -85,B 0,C 180,E1 -10268.695,E2 -10268.695} C_VEL
LIN {X 0,Y 418.322,Z 379.379,A -85,B 0,C 180,E1 -10271.631,E2 -10271.631} C_VEL
LIN {X 0,Y 418.309,Z 379.377,A -85,B 0,C 180,E1 -10274.597,E2 -10274.597} C_VEL
LIN {X 0,Y 418.294,Z 379.383,A -85,B 0,C 180,E1 -10277.604,E2 -10277.604} C_VEL
LIN {X 0,Y 418.256,Z 379.384,A -85,B 0,C 180,E1 -10280.663,E2 -10280.663} C_VEL
LIN {X 0,Y 418.292,Z 379.38,A -85,B 0,C 180,E1 -10283.781,E2 -10283.781} C_VEL
LIN {X 0,Y 418.326,Z 379.377,A -85,B 0,C 180,E1 -10287.073,E2 -10287.073} C_VEL
LIN {X 0,Y 418.332,Z 379.496,A -85,B 0,C 180,E1 -10288.163,E2 -10288.163} C_VEL
LIN {X 0,Y 420.175,Z 389.1,A -85,B 0,C 180,E1 -10290.674,E2 -10290.674} C_VEL
LIN {X 0,Y 420.499,Z 392.497,A -85,B 0,C 180,E1 -10291.526,E2 -10291.526} C_VEL
LIN {X 0,Y 420.229,Z 398.362,A -85,B 0,C 180,E1 -10292.902,E2 -10292.902} C_VEL
LIN {X 0,Y 424.215,Z 417.47,A -85,B 0,C 180,E1 -10293.462,E2 -10293.462} C_VEL
LIN {X 0,Y 423.002,Z 505.298,A -85,B 0,C 180,E1 -10295.047,E2 -10295.047} C_VEL
LIN {X 0,Y 422.588,Z 518.314,A -85,B 0,C 180,E1 -10295.469,E2 -10295.469} C_VEL
LIN {X 0,Y 422.051,Z 531.244,A -85,B 0,C 180,E1 -10296.091,E2 -10296.091} C_VEL
LIN {X 0,Y 421.434,Z 542.488,A -85,B 0,C 180,E1 -10296.824,E2 -10296.824} C_VEL
LIN {X 0,Y 420.749,Z 553.229,A -85,B 0,C 180,E1 -10297.717,E2 -10297.717} C_VEL
LIN {X 0,Y 419.954,Z 564.326,A -85,B 0,C 180,E1 -10298.871,E2 -10298.871} C_VEL
LIN {X 0,Y 419.231,Z 573.378,A -85,B 0,C 180,E1 -10300.04,E2 -10300.04} C_VEL
LIN {X 0,Y 418.658,Z 580.87,A -85,B 0,C 180,E1 -10301.215,E2 -10301.215} C_VEL
LIN {X 0,Y 418.137,Z 588.386,A -85,B 0,C 180,E1 -10302.662,E2 -10302.662} C_VEL
LIN {X 0,Y 417.643,Z 595.304,A -85,B 0,C 180,E1 -10304.341,E2 -10304.341} C_VEL
LIN {X 0,Y 417.382,Z 599.567,A -85,B 0,C 180,E1 -10305.669,E2 -10305.669} C_VEL
LIN {X 0,Y 417.174,Z 602.961,A -85,B 0,C 180,E1 -10307.018,E2 -10307.018} C_VEL
LIN {X 0,Y 416.956,Z 606.273,A -85,B 0,C 180,E1 -10308.9,E2 -10308.9} C_VEL
LIN {X 0,Y 416.833,Z 607.993,A -85,B 0,C 180,E1 -10310.858,E2 -10310.858} C_VEL
LIN {X 0,Y 416.872,Z 608.163,A -85,B 0,C 180,E1 -10312.632,E2 -10312.632} C_VEL
LIN {X 0,Y 416.87,Z 607.335,A -85,B 0,C 180,E1 -10314.021,E2 -10314.021} C_VEL
LIN {X 0,Y 417.001,Z 605.278,A -85,B 0,C 180,E1 -10315.673,E2 -10315.673} C_VEL
LIN {X 0,Y 417.244,Z 601.843,A -85,B 0,C 180,E1 -10317.383,E2 -10317.383} C_VEL
LIN {X 0,Y 417.508,Z 596.734,A -85,B 0,C 180,E1 -10319.148,E2 -10319.148} C_VEL
LIN {X 0,Y 417.912,Z 590.362,A -85,B 0,C 180,E1 -10320.81,E2 -10320.81} C_VEL
LIN {X 0,Y 418.374,Z 583.67,A -85,B 0,C 180,E1 -10322.186,E2 -10322.186} C_VEL
LIN {X 0,Y 418.941,Z 575.106,A -85,B 0,C 180,E1 -10323.604,E2 -10323.604} C_VEL
LIN {X 0,Y 419.634,Z 565.364,A -85,B 0,C 180,E1 -10324.908,E2 -10324.908} C_VEL
LIN {X 0,Y 420.33,Z 555.764,A -85,B 0,C 180,E1 -10325.948,E2 -10325.948} C_VEL
LIN {X 0,Y 420.99,Z 543.806,A -85,B 0,C 180,E1 -10326.98,E2 -10326.98} C_VEL
LIN {X 0,Y 421.669,Z 531.828,A -85,B 0,C 180,E1 -10327.781,E2 -10327.781} C_VEL
LIN {X 0,Y 422.148,Z 519.329,A -85,B 0,C 180,E1 -10328.402,E2 -10328.402} C_VEL
LIN {X 0,Y 422.606,Z 505.291,A -85,B 0,C 180,E1 -10328.866,E2 -10328.866} C_VEL
LIN {X 0,Y 423.484,Z 441.365,A -85,B 0,C 180,E1 -10330.011,E2 -10330.011} C_VEL
LIN {X 0,Y 422.993,Z 435.548,A -85,B 0,C 180,E1 -10330.138,E2 -10330.138} C_VEL
LIN {X 0,Y 420.321,Z 426.23,A -85,B 0,C 180,E1 -10330.423,E2 -10330.423} C_VEL
LIN {X 0,Y 416.502,Z 415.115,A -85,B 0,C 180,E1 -10330.795,E2 -10330.795} C_VEL
LIN {X 0,Y 415.641,Z 411.28,A -85,B 0,C 180,E1 -10330.904,E2 -10330.904} C_VEL
LIN {X 0,Y 412.947,Z 397.717,A -85,B 0,C 180,E1 -10331.293,E2 -10331.293} C_VEL
LIN {X 0,Y 413.287,Z 391.672,A -85,B 0,C 180,E1 -10332.726,E2 -10332.726} C_VEL
LIN {X 0,Y 411.391,Z 380.653,A -85,B 0,C 180,E1 -10335.53,E2 -10335.53} C_VEL
LIN {X 0,Y 411.308,Z 380.252,A -85,B 0,C 180,E1 -10335.654,E2 -10335.654} C_VEL
LIN {X 0,Y 411.292,Z 380.252,A -85,B 0,C 180,E1 -10339.165,E2 -10339.165} C_VEL
LIN {X 0,Y 411.402,Z 380.239,A -85,B 0,C 180,E1 -10342.232,E2 -10342.232} C_VEL
LIN {X 0,Y 411.448,Z 380.233,A -85,B 0,C 180,E1 -10344.116,E2 -10344.116} C_VEL
LIN {X 0,Y 411.516,Z 380.224,A -85,B 0,C 180,E1 -10348.041,E2 -10348.041} C_VEL
LIN {X 0,Y 411.644,Z 380.208,A -85,B 0,C 180,E1 -10349.999,E2 -10349.999} C_VEL
LIN {X 0,Y 411.469,Z 380.227,A -85,B 0,C 180,E1 -10352.936,E2 -10352.936} C_VEL
LIN {X 0,Y 411.463,Z 380.228,A -85,B 0,C 180,E1 -10356.866,E2 -10356.866} C_VEL
LIN {X 0,Y 411.294,Z 380.252,A -85,B 0,C 180,E1 -10359.837,E2 -10359.837} C_VEL
LIN {X 0,Y 411.307,Z 380.247,A -85,B 0,C 180,E1 -10363.103,E2 -10363.103} C_VEL
LIN {X 0,Y 411.265,Z 380.252,A -85,B 0,C 180,E1 -10366.868,E2 -10366.868} C_VEL
LIN {X 0,Y 411.23,Z 380.263,A -85,B 0,C 180,E1 -10369.985,E2 -10369.985} C_VEL
LIN {X 0,Y 411.194,Z 380.261,A -85,B 0,C 180,E1 -10373.146,E2 -10373.146} C_VEL
LIN {X 0,Y 411.235,Z 380.257,A -85,B 0,C 180,E1 -10376.379,E2 -10376.379} C_VEL
LIN {X 0,Y 411.231,Z 380.263,A -85,B 0,C 180,E1 -10379.709,E2 -10379.709} C_VEL
LIN {X 0,Y 411.203,Z 380.261,A -85,B 0,C 180,E1 -10383.154,E2 -10383.154} C_VEL
LIN {X 0,Y 411.192,Z 380.261,A -85,B 0,C 180,E1 -10386.552,E2 -10386.552} C_VEL
LIN {X 0,Y 411.223,Z 380.263,A -85,B 0,C 180,E1 -10389.729,E2 -10389.729} C_VEL
LIN {X 0,Y 411.176,Z 380.266,A -85,B 0,C 180,E1 -10393.131,E2 -10393.131} C_VEL
LIN {X 0,Y 411.284,Z 380.349,A -85,B 0,C 180,E1 -10395.543,E2 -10395.543} C_VEL
LIN {X 0,Y 412.834,Z 388.935,A -85,B 0,C 180,E1 -10397.4,E2 -10397.4} C_VEL
LIN {X 0,Y 412.655,Z 396.445,A -85,B 0,C 180,E1 -10398.95,E2 -10398.95} C_VEL
LIN {X 0,Y 416.587,Z 418.651,A -85,B 0,C 180,E1 -10399.574,E2 -10399.574} C_VEL
LIN {X 0,Y 415.186,Z 505.112,A -85,B 0,C 180,E1 -10401.26,E2 -10401.26} C_VEL
LIN {X 0,Y 414.75,Z 518.603,A -85,B 0,C 180,E1 -10401.716,E2 -10401.716} C_VEL
LIN {X 0,Y 414.244,Z 531.29,A -85,B 0,C 180,E1 -10402.354,E2 -10402.354} C_VEL
LIN {X 0,Y 413.604,Z 543.86,A -85,B 0,C 180,E1 -10403.201,E2 -10403.201} C_VEL
LIN {X 0,Y 412.941,Z 555.194,A -85,B 0,C 180,E1 -10404.194,E2 -10404.194} C_VEL
LIN {X 0,Y 412.291,Z 565.581,A -85,B 0,C 180,E1 -10405.325,E2 -10405.325} C_VEL
LIN {X 0,Y 411.637,Z 575.154,A -85,B 0,C 180,E1 -10406.62,E2 -10406.62} C_VEL
LIN {X 0,Y 411.15,Z 583.43,A -85,B 0,C 180,E1 -10408.001,E2 -10408.001} C_VEL
LIN {X 0,Y 410.691,Z 590.234,A -85,B 0,C 180,E1 -10409.396,E2 -10409.396} C_VEL
LIN {X 0,Y 410.354,Z 595.973,A -85,B 0,C 180,E1 -10410.86,E2 -10410.86} C_VEL
LIN {X 0,Y 410.122,Z 600.764,A -85,B 0,C 180,E1 -10412.439,E2 -10412.439} C_VEL
LIN {X 0,Y 409.976,Z 604.409,A -85,B 0,C 180,E1 -10414.079,E2 -10414.079} C_VEL
LIN {X 0,Y 409.825,Z 606.799,A -85,B 0,C 180,E1 -10415.696,E2 -10415.696} C_VEL
LIN {X 0,Y 409.749,Z 607.765,A -85,B 0,C 180,E1 -10416.765,E2 -10416.765} C_VEL
LIN {X 0,Y 409.738,Z 608.199,A -85,B 0,C 180,E1 -10417.85,E2 -10417.85} C_VEL
LIN {X 0,Y 409.762,Z 608.179,A -85,B 0,C 180,E1 -10418.889,E2 -10418.889} C_VEL
LIN {X 0,Y 409.841,Z 607.13,A -85,B 0,C 180,E1 -10420.581,E2 -10420.581} C_VEL
LIN {X 0,Y 409.957,Z 605.25,A -85,B 0,C 180,E1 -10422.026,E2 -10422.026} C_VEL
LIN {X 0,Y 410.182,Z 602.036,A -85,B 0,C 180,E1 -10423.631,E2 -10423.631} C_VEL
LIN {X 0,Y 410.408,Z 597.951,A -85,B 0,C 180,E1 -10425.116,E2 -10425.116} C_VEL
LIN {X 0,Y 410.858,Z 592.253,A -85,B 0,C 180,E1 -10426.699,E2 -10426.699} C_VEL
LIN {X 0,Y 411.333,Z 585.579,A -85,B 0,C 180,E1 -10428.169,E2 -10428.169} C_VEL
LIN {X 0,Y 411.883,Z 578.542,A -85,B 0,C 180,E1 -10429.43,E2 -10429.43} C_VEL
LIN {X 0,Y 412.641,Z 568.999,A -85,B 0,C 180,E1 -10430.82,E2 -10430.82} C_VEL
LIN {X 0,Y 413.424,Z 558.43,A -85,B 0,C 180,E1 -10432.061,E2 -10432.061} C_VEL
LIN {X 0,Y 414.193,Z 547.787,A -85,B 0,C 180,E1 -10433.056,E2 -10433.056} C_VEL
LIN {X 0,Y 414.924,Z 536.068,A -85,B 0,C 180,E1 -10433.923,E2 -10433.923} C_VEL
LIN {X 0,Y 415.488,Z 524.198,A -85,B 0,C 180,E1 -10434.601,E2 -10434.601} C_VEL
LIN {X 0,Y 415.972,Z 511.301,A -85,B 0,C 180,E1 -10435.124,E2 -10435.124} C_VEL
LIN {X 0,Y 416.325,Z 497.226,A -85,B 0,C 180,E1 -10435.481,E2 -10435.481} C_VEL
LIN {X 0,Y 417.793,Z 418.045,A -85,B 0,C 180,E1 -10437.079,E2 -10437.079} C_VEL
LIN {X 0,Y 414.799,Z 403.21,A -85,B 0,C 180,E1 -10437.588,E2 -10437.588} C_VEL
LIN {X 0,Y 413.463,Z 397.344,A -85,B 0,C 180,E1 -10437.808,E2 -10437.808} C_VEL
LIN {X 0,Y 413.438,Z 390.211,A -85,B 0,C 180,E1 -10439.269,E2 -10439.269} C_VEL
LIN {X 0,Y 412.209,Z 383.403,A -85,B 0,C 180,E1 -10440.733,E2 -10440.733} C_VEL
LIN {X 0,Y 411.483,Z 380.231,A -85,B 0,C 180,E1 -10441.468,E2 -10441.468} C_VEL
LIN {X 0,Y 411.457,Z 380.237,A -85,B 0,C 180,E1 -10442.937,E2 -10442.937} C_VEL
LIN {X 0,Y 411.449,Z 380.235,A -85,B 0,C 180,E1 -10446.867,E2 -10446.867} C_VEL
LIN {X 0,Y 411.298,Z 380.253,A -85,B 0,C 180,E1 -10449.839,E2 -10449.839} C_VEL
LIN {X 0,Y 411.302,Z 380.251,A -85,B 0,C 180,E1 -10453.109,E2 -10453.109} C_VEL
LIN {X 0,Y 411.252,Z 380.257,A -85,B 0,C 180,E1 -10456.889,E2 -10456.889} C_VEL
LIN {X 0,Y 411.245,Z 380.26,A -85,B 0,C 180,E1 -10459.986,E2 -10459.986} C_VEL
LIN {X 0,Y 411.221,Z 380.259,A -85,B 0,C 180,E1 -10463.146,E2 -10463.146} C_VEL
LIN {X 0,Y 411.23,Z 380.26,A -85,B 0,C 180,E1 -10466.381,E2 -10466.381} C_VEL
LIN {X 0,Y 411.202,Z 380.265,A -85,B 0,C 180,E1 -10469.713,E2 -10469.713} C_VEL
LIN {X 0,Y 411.198,Z 380.265,A -85,B 0,C 180,E1 -10473.157,E2 -10473.157} C_VEL
LIN {X 0,Y 411.187,Z 380.264,A -85,B 0,C 180,E1 -10476.554,E2 -10476.554} C_VEL
LIN {X 0,Y 411.211,Z 380.264,A -85,B 0,C 180,E1 -10479.73,E2 -10479.73} C_VEL
LIN {X 0,Y 411.17,Z 380.269,A -85,B 0,C 180,E1 -10483.134,E2 -10483.134} C_VEL
LIN {X 0,Y 411.167,Z 380.266,A -85,B 0,C 180,E1 -10485.881,E2 -10485.881} C_VEL
LIN {X 0,Y 411.158,Z 380.27,A -85,B 0,C 180,E1 -10488.773,E2 -10488.773} C_VEL
LIN {X 0,Y 411.195,Z 380.263,A -85,B 0,C 180,E1 -10492.028,E2 -10492.028} C_VEL
LIN {X 0,Y 411.202,Z 380.263,A -85,B 0,C 180,E1 -10495.668,E2 -10495.668} C_VEL
LIN {X 0,Y 411.199,Z 380.265,A -85,B 0,C 180,E1 -10499.155,E2 -10499.155} C_VEL
LIN {X 0,Y 411.302,Z 380.273,A -85,B 0,C 180,E1 -10502.389,E2 -10502.389} C_VEL
LIN {X 0,Y 413.893,Z 393.644,A -85,B 0,C 180,E1 -10505.418,E2 -10505.418} C_VEL
LIN {X 0,Y 414.25,Z 396.179,A -85,B 0,C 180,E1 -10505.974,E2 -10505.974} C_VEL
LIN {X 0,Y 413.379,Z 410.038,A -85,B 0,C 180,E1 -10508.823,E2 -10508.823} C_VEL
LIN {X 0,Y 412.837,Z 418.325,A -85,B 0,C 180,E1 -10510.485,E2 -10510.485} C_VEL
LIN {X 0,Y 415.763,Z 436.805,A -85,B 0,C 180,E1 -10511.071,E2 -10511.071} C_VEL
LIN {X 0,Y 416.91,Z 446.349,A -85,B 0,C 180,E1 -10511.348,E2 -10511.348} C_VEL
LIN {X 0,Y 416.305,Z 484.804,A -85,B 0,C 180,E1 -10512.106,E2 -10512.106} C_VEL
LIN {X 0,Y 415.708,Z 528.709,A -85,B 0,C 180,E1 -10512.919,E2 -10512.919} C_VEL
LIN {X 0,Y 415.113,Z 542.204,A -85,B 0,C 180,E1 -10513.369,E2 -10513.369} C_VEL
LIN {X 0,Y 414.513,Z 554.98,A -85,B 0,C 180,E1 -10514.009,E2 -10514.009} C_VEL
LIN {X 0,Y 413.729,Z 567.497,A -85,B 0,C 180,E1 -10514.862,E2 -10514.862} C_VEL
LIN {X 0,Y 412.947,Z 578.847,A -85,B 0,C 180,E1 -10515.856,E2 -10515.856} C_VEL
LIN {X 0,Y 412.255,Z 588.748,A -85,B 0,C 180,E1 -10516.947,E2 -10516.947} C_VEL
LIN {X 0,Y 411.626,Z 597.859,A -85,B 0,C 180,E1 -10518.179,E2 -10518.179} C_VEL
LIN {X 0,Y 410.97,Z 606.747,A -85,B 0,C 180,E1 -10519.657,E2 -10519.657} C_VEL
LIN {X 0,Y 410.532,Z 613.855,A -85,B 0,C 180,E1 -10521.138,E2 -10521.138} C_VEL
LIN {X 0,Y 410.2,Z 619.525,A -85,B 0,C 180,E1 -10522.619,E2 -10522.619} C_VEL
LIN {X 0,Y 410.035,Z 623.98,A -85,B 0,C 180,E1 -10524.099,E2 -10524.099} C_VEL
LIN {X 0,Y 410.019,Z 626.331,A -85,B 0,C 180,E1 -10525.085,E2 -10525.085} C_VEL
LIN {X 0,Y 409.932,Z 628.245,A -85,B 0,C 180,E1 -10526.069,E2 -10526.069} C_VEL
LIN {X 0,Y 409.926,Z 629.706,A -85,B 0,C 180,E1 -10527.053,E2 -10527.053} C_VEL
LIN {X 0,Y 409.966,Z 630.734,A -85,B 0,C 180,E1 -10528.036,E2 -10528.036} C_VEL
LIN {X 0,Y 409.935,Z 631.366,A -85,B 0,C 180,E1 -10529.019,E2 -10529.019} C_VEL
LIN {X 0,Y 409.926,Z 631.607,A -85,B 0,C 180,E1 -10530.001,E2 -10530.001} C_VEL
LIN {X 0,Y 409.935,Z 631.421,A -85,B 0,C 180,E1 -10530.984,E2 -10530.984} C_VEL
LIN {X 0,Y 409.967,Z 630.819,A -85,B 0,C 180,E1 -10531.966,E2 -10531.966} C_VEL
LIN {X 0,Y 409.932,Z 628.427,A -85,B 0,C 180,E1 -10533.934,E2 -10533.934} C_VEL
LIN {X 0,Y 410.021,Z 625.483,A -85,B 0,C 180,E1 -10535.411,E2 -10535.411} C_VEL
LIN {X 0,Y 410.168,Z 621.5,A -85,B 0,C 180,E1 -10536.89,E2 -10536.89} C_VEL
LIN {X 0,Y 410.48,Z 615.383,A -85,B 0,C 180,E1 -10538.617,E2 -10538.617} C_VEL
LIN {X 0,Y 410.916,Z 608.688,A -85,B 0,C 180,E1 -10540.098,E2 -10540.098} C_VEL
LIN {X 0,Y 411.526,Z 600.385,A -85,B 0,C 180,E1 -10541.577,E2 -10541.577} C_VEL
LIN {X 0,Y 412.268,Z 591.895,A -85,B 0,C 180,E1 -10542.805,E2 -10542.805} C_VEL
LIN {X 0,Y 412.955,Z 581.263,A -85,B 0,C 180,E1 -10544.053,E2 -10544.053} C_VEL
LIN {X 0,Y 413.824,Z 569.633,A -85,B 0,C 180,E1 -10545.137,E2 -10545.137} C_VEL
LIN {X 0,Y 414.637,Z 557.863,A -85,B 0,C 180,E1 -10545.989,E2 -10545.989} C_VEL
LIN {X 0,Y 415.418,Z 544.381,A -85,B 0,C 180,E1 -10546.716,E2 -10546.716} C_VEL
LIN {X 0,Y 415.952,Z 532.425,A -85,B 0,C 180,E1 -10547.168,E2 -10547.168} C_VEL
LIN {X 0,Y 416.39,Z 517.751,A -85,B 0,C 180,E1 -10547.498,E2 -10547.498} C_VEL
LIN {X 0,Y 417.198,Z 444.859,A -85,B 0,C 180,E1 -10548.824,E2 -10548.824} C_VEL
LIN {X 0,Y 412.903,Z 418.718,A -85,B 0,C 180,E1 -10549.561,E2 -10549.561} C_VEL
LIN {X 0,Y 414.117,Z 402.186,A -85,B 0,C 180,E1 -10552.976,E2 -10552.976} C_VEL
LIN {X 0,Y 414.418,Z 395.997,A -85,B 0,C 180,E1 -10554.284,E2 -10554.284} C_VEL
LIN {X 0,Y 412.281,Z 384.91,A -85,B 0,C 180,E1 -10556.856,E2 -10556.856} C_VEL
LIN {X 0,Y 411.27,Z 380.262,A -85,B 0,C 180,E1 -10557.997,E2 -10557.997} C_VEL
LIN {X 0,Y 411.188,Z 380.271,A -85,B 0,C 180,E1 -10561.284,E2 -10561.284} C_VEL
LIN {X 0,Y 411.211,Z 380.261,A -85,B 0,C 180,E1 -10564.334,E2 -10564.334} C_VEL
LIN {X 0,Y 411.201,Z 380.265,A -85,B 0,C 180,E1 -10567.974,E2 -10567.974} C_VEL
LIN {X 0,Y 411.187,Z 380.268,A -85,B 0,C 180,E1 -10570.505,E2 -10570.505} C_VEL
LIN {X 0,Y 411.179,Z 380.272,A -85,B 0,C 180,E1 -10573.134,E2 -10573.134} C_VEL
LIN {X 0,Y 411.174,Z 380.267,A -85,B 0,C 180,E1 -10575.882,E2 -10575.882} C_VEL
LIN {X 0,Y 411.169,Z 380.271,A -85,B 0,C 180,E1 -10578.772,E2 -10578.772} C_VEL
LIN {X 0,Y 411.198,Z 380.262,A -85,B 0,C 180,E1 -10582.027,E2 -10582.027} C_VEL
LIN {X 0,Y 411.211,Z 380.257,A -85,B 0,C 180,E1 -10585.667,E2 -10585.667} C_VEL
LIN {X 0,Y 411.195,Z 380.258,A -85,B 0,C 180,E1 -10589.153,E2 -10589.153} C_VEL
LIN {X 0,Y 411.265,Z 380.255,A -85,B 0,C 180,E1 -10592.523,E2 -10592.523} C_VEL
LIN {X 0,Y 411.231,Z 380.258,A -85,B 0,C 180,E1 -10595.785,E2 -10595.785} C_VEL
LIN {X 0,Y 411.202,Z 380.264,A -85,B 0,C 180,E1 -10598.966,E2 -10598.966} C_VEL
LIN {X 0,Y 411.258,Z 380.251,A -85,B 0,C 180,E1 -10602.085,E2 -10602.085} C_VEL
LIN {X 0,Y 411.266,Z 380.247,A -85,B 0,C 180,E1 -10605.148,E2 -10605.148} C_VEL
LIN {X 0,Y 411.29,Z 380.255,A -85,B 0,C 180,E1 -10608.167,E2 -10608.167} C_VEL
LIN {X 0,Y 411.488,Z 380.229,A -85,B 0,C 180,E1 -10612.147,E2 -10612.147} C_VEL
LIN {X 0,Y 411.481,Z 380.226,A -85,B 0,C 180,E1 -10614.118,E2 -10614.118} C_VEL
LIN {X 0,Y 411.517,Z 380.223,A -85,B 0,C 180,E1 -10618.043,E2 -10618.043} C_VEL
LIN {X 0,Y 411.646,Z 380.208,A -85,B 0,C 180,E1 -10620,E2 -10620} C_VEL
LIN {X 0,Y 411.464,Z 380.228,A -85,B 0,C 180,E1 -10622.937,E2 -10622.937} C_VEL
LIN {X 0,Y 411.467,Z 380.226,A -85,B 0,C 180,E1 -10626.867,E2 -10626.867} C_VEL
LIN {X 0,Y 411.361,Z 380.242,A -85,B 0,C 180,E1 -10628.845,E2 -10628.845} C_VEL
LIN {X 0,Y 411.29,Z 380.254,A -85,B 0,C 180,E1 -10631.833,E2 -10631.833} C_VEL
LIN {X 0,Y 411.266,Z 380.254,A -85,B 0,C 180,E1 -10634.853,E2 -10634.853} C_VEL
LIN {X 0,Y 411.259,Z 380.259,A -85,B 0,C 180,E1 -10637.915,E2 -10637.915} C_VEL
LIN {X 0,Y 411.203,Z 380.264,A -85,B 0,C 180,E1 -10641.034,E2 -10641.034} C_VEL
LIN {X 0,Y 411.232,Z 380.261,A -85,B 0,C 180,E1 -10644.215,E2 -10644.215} C_VEL
LIN {X 0,Y 411.276,Z 380.367,A -85,B 0,C 180,E1 -10647.857,E2 -10647.857} C_VEL
LIN {X 0,Y 413.124,Z 389.892,A -85,B 0,C 180,E1 -10650.404,E2 -10650.404} C_VEL
LIN {X 0,Y 413.579,Z 394.183,A -85,B 0,C 180,E1 -10651.503,E2 -10651.503} C_VEL
LIN {X 0,Y 413.351,Z 398.389,A -85,B 0,C 180,E1 -10652.527,E2 -10652.527} C_VEL
LIN {X 0,Y 417.606,Z 418.949,A -85,B 0,C 180,E1 -10653.159,E2 -10653.159} C_VEL
LIN {X 0,Y 416.241,Z 505.914,A -85,B 0,C 180,E1 -10654.758,E2 -10654.758} C_VEL
LIN {X 0,Y 415.796,Z 519.643,A -85,B 0,C 180,E1 -10655.222,E2 -10655.222} C_VEL
LIN {X 0,Y 415.214,Z 532.556,A -85,B 0,C 180,E1 -10655.875,E2 -10655.875} C_VEL
LIN {X 0,Y 414.556,Z 543.857,A -85,B 0,C 180,E1 -10656.643,E2 -10656.643} C_VEL
LIN {X 0,Y 413.841,Z 554.175,A -85,B 0,C 180,E1 -10657.529,E2 -10657.529} C_VEL
LIN {X 0,Y 413.032,Z 565.141,A -85,B 0,C 180,E1 -10658.704,E2 -10658.704} C_VEL
LIN {X 0,Y 412.242,Z 574.113,A -85,B 0,C 180,E1 -10659.898,E2 -10659.898} C_VEL
LIN {X 0,Y 411.565,Z 582.599,A -85,B 0,C 180,E1 -10661.291,E2 -10661.291} C_VEL
LIN {X 0,Y 411.056,Z 589.458,A -85,B 0,C 180,E1 -10662.676,E2 -10662.676} C_VEL
LIN {X 0,Y 410.655,Z 594.965,A -85,B 0,C 180,E1 -10664.044,E2 -10664.044} C_VEL
LIN {X 0,Y 410.359,Z 599.349,A -85,B 0,C 180,E1 -10665.396,E2 -10665.396} C_VEL
LIN {X 0,Y 410.12,Z 602.76,A -85,B 0,C 180,E1 -10666.727,E2 -10666.727} C_VEL
LIN {X 0,Y 409.935,Z 605.315,A -85,B 0,C 180,E1 -10668.038,E2 -10668.038} C_VEL
LIN {X 0,Y 409.827,Z 607.05,A -85,B 0,C 180,E1 -10669.333,E2 -10669.333} C_VEL
LIN {X 0,Y 409.742,Z 608.091,A -85,B 0,C 180,E1 -10670.606,E2 -10670.606} C_VEL
LIN {X 0,Y 409.759,Z 608.46,A -85,B 0,C 180,E1 -10672.09,E2 -10672.09} C_VEL
LIN {X 0,Y 409.76,Z 607.802,A -85,B 0,C 180,E1 -10673.719,E2 -10673.719} C_VEL
LIN {X 0,Y 409.887,Z 605.748,A -85,B 0,C 180,E1 -10675.539,E2 -10675.539} C_VEL
LIN {X 0,Y 410.102,Z 602.82,A -85,B 0,C 180,E1 -10677.111,E2 -10677.111} C_VEL
LIN {X 0,Y 410.383,Z 598.089,A -85,B 0,C 180,E1 -10678.901,E2 -10678.901} C_VEL
LIN {X 0,Y 410.755,Z 592.23,A -85,B 0,C 180,E1 -10680.537,E2 -10680.537} C_VEL
LIN {X 0,Y 411.212,Z 585.779,A -85,B 0,C 180,E1 -10681.964,E2 -10681.964} C_VEL
LIN {X 0,Y 411.764,Z 577.878,A -85,B 0,C 180,E1 -10683.381,E2 -10683.381} C_VEL
LIN {X 0,Y 412.401,Z 569.666,A -85,B 0,C 180,E1 -10684.584,E2 -10684.584} C_VEL
LIN {X 0,Y 413.167,Z 559.723,A -85,B 0,C 180,E1 -10685.771,E2 -10685.771} C_VEL
LIN {X 0,Y 413.859,Z 548.37,A -85,B 0,C 180,E1 -10686.857,E2 -10686.857} C_VEL
LIN {X 0,Y 414.61,Z 536.051,A -85,B 0,C 180,E1 -10687.776,E2 -10687.776} C_VEL
LIN {X 0,Y 415.106,Z 525.154,A -85,B 0,C 180,E1 -10688.396,E2 -10688.396} C_VEL
LIN {X 0,Y 415.587,Z 511.331,A -85,B 0,C 180,E1 -10688.958,E2 -10688.958} C_VEL
LIN {X 0,Y 415.913,Z 498.487,A -85,B 0,C 180,E1 -10689.279,E2 -10689.279} C_VEL
LIN {X 0,Y 416.974,Z 418.413,A -85,B 0,C 180,E1 -10690.712,E2 -10690.712} C_VEL
LIN {X 0,Y 415.641,Z 411.28,A -85,B 0,C 180,E1 -10690.904,E2 -10690.904} C_VEL
LIN {X 0,Y 414.739,Z 407.673,A -85,B 0,C 180,E1 -10691.048,E2 -10691.048} C_VEL
LIN {X 0,Y 412.731,Z 402.836,A -85,B 0,C 180,E1 -10691.399,E2 -10691.399} C_VEL
LIN {X 0,Y 409.625,Z 397.399,A -85,B 0,C 180,E1 -10692.06,E2 -10692.06} C_VEL
LIN {X 0,Y 406.93,Z 392.817,A -85,B 0,C 180,E1 -10692.895,E2 -10692.895} C_VEL
LIN {X 0,Y 405.847,Z 389.804,A -85,B 0,C 180,E1 -10693.605,E2 -10693.605} C_VEL
LIN {X 0,Y 404.251,Z 381.131,A -85,B 0,C 180,E1 -10695.912,E2 -10695.912} C_VEL
LIN {X 0,Y 404.258,Z 381.13,A -85,B 0,C 180,E1 -10698.974,E2 -10698.974} C_VEL
LIN {X 0,Y 404.365,Z 381.115,A -85,B 0,C 180,E1 -10702.173,E2 -10702.173} C_VEL
LIN {X 0,Y 404.281,Z 381.123,A -85,B 0,C 180,E1 -10705.012,E2 -10705.012} C_VEL
LIN {X 0,Y 404.485,Z 381.1,A -85,B 0,C 180,E1 -10708.007,E2 -10708.007} C_VEL
LIN {X 0,Y 404.614,Z 381.084,A -85,B 0,C 180,E1 -10709.999,E2 -10709.999} C_VEL
LIN {X 0,Y 404.426,Z 381.105,A -85,B 0,C 180,E1 -10712.987,E2 -10712.987} C_VEL
LIN {X 0,Y 404.415,Z 381.106,A -85,B 0,C 180,E1 -10716.986,E2 -10716.986} C_VEL
LIN {X 0,Y 404.26,Z 381.13,A -85,B 0,C 180,E1 -10720.01,E2 -10720.01} C_VEL
LIN {X 0,Y 404.267,Z 381.124,A -85,B 0,C 180,E1 -10723.21,E2 -10723.21} C_VEL
LIN {X 0,Y 404.219,Z 381.13,A -85,B 0,C 180,E1 -10727.007,E2 -10727.007} C_VEL
LIN {X 0,Y 404.163,Z 381.139,A -85,B 0,C 180,E1 -10730.35,E2 -10730.35} C_VEL
LIN {X 0,Y 404.162,Z 381.14,A -85,B 0,C 180,E1 -10733.573,E2 -10733.573} C_VEL
LIN {X 0,Y 404.181,Z 381.141,A -85,B 0,C 180,E1 -10735.765,E2 -10735.765} C_VEL
LIN {X 0,Y 404.196,Z 381.137,A -85,B 0,C 180,E1 -10737.998,E2 -10737.998} C_VEL
LIN {X 0,Y 404.148,Z 381.142,A -85,B 0,C 180,E1 -10741.444,E2 -10741.444} C_VEL
LIN {X 0,Y 404.182,Z 381.135,A -85,B 0,C 180,E1 -10745.014,E2 -10745.014} C_VEL
LIN {X 0,Y 404.159,Z 381.137,A -85,B 0,C 180,E1 -10748.754,E2 -10748.754} C_VEL
LIN {X 0,Y 404.145,Z 381.145,A -85,B 0,C 180,E1 -10751.603,E2 -10751.603} C_VEL
LIN {X 0,Y 404.227,Z 381.187,A -85,B 0,C 180,E1 -10755.366,E2 -10755.366} C_VEL
LIN {X 0,Y 405.888,Z 391.09,A -85,B 0,C 180,E1 -10757.523,E2 -10757.523} C_VEL
LIN {X 0,Y 405.721,Z 396.536,A -85,B 0,C 180,E1 -10758.651,E2 -10758.651} C_VEL
LIN {X 0,Y 409.762,Z 419.666,A -85,B 0,C 180,E1 -10759.326,E2 -10759.326} C_VEL
LIN {X 0,Y 408.289,Z 505.487,A -85,B 0,C 180,E1 -10761.036,E2 -10761.036} C_VEL
LIN {X 0,Y 407.831,Z 518.859,A -85,B 0,C 180,E1 -10761.499,E2 -10761.499} C_VEL
LIN {X 0,Y 407.334,Z 531.423,A -85,B 0,C 180,E1 -10762.143,E2 -10762.143} C_VEL
LIN {X 0,Y 406.709,Z 543.191,A -85,B 0,C 180,E1 -10762.94,E2 -10762.94} C_VEL
LIN {X 0,Y 406.002,Z 554.68,A -85,B 0,C 180,E1 -10763.946,E2 -10763.946} C_VEL
LIN {X 0,Y 405.329,Z 565.192,A -85,B 0,C 180,E1 -10765.097,E2 -10765.097} C_VEL
LIN {X 0,Y 404.726,Z 573.765,A -85,B 0,C 180,E1 -10766.242,E2 -10766.242} C_VEL
LIN {X 0,Y 404.17,Z 582.493,A -85,B 0,C 180,E1 -10767.676,E2 -10767.676} C_VEL
LIN {X 0,Y 403.698,Z 589.507,A -85,B 0,C 180,E1 -10769.098,E2 -10769.098} C_VEL
LIN {X 0,Y 403.286,Z 596.173,A -85,B 0,C 180,E1 -10770.794,E2 -10770.794} C_VEL
LIN {X 0,Y 403.05,Z 600.969,A -85,B 0,C 180,E1 -10772.403,E2 -10772.403} C_VEL
LIN {X 0,Y 402.87,Z 604.747,A -85,B 0,C 180,E1 -10774.143,E2 -10774.143} C_VEL
LIN {X 0,Y 402.767,Z 606.456,A -85,B 0,C 180,E1 -10775.242,E2 -10775.242} C_VEL
LIN {X 0,Y 402.666,Z 607.594,A -85,B 0,C 180,E1 -10776.332,E2 -10776.332} C_VEL
LIN {X 0,Y 402.644,Z 608.351,A -85,B 0,C 180,E1 -10777.678,E2 -10777.678} C_VEL
LIN {X 0,Y 402.685,Z 608.12,A -85,B 0,C 180,E1 -10779.57,E2 -10779.57} C_VEL
LIN {X 0,Y 402.757,Z 607.355,A -85,B 0,C 180,E1 -10780.637,E2 -10780.637} C_VEL
LIN {X 0,Y 402.824,Z 606.081,A -85,B 0,C 180,E1 -10781.697,E2 -10781.697} C_VEL
LIN {X 0,Y 403.087,Z 602.793,A -85,B 0,C 180,E1 -10783.52,E2 -10783.52} C_VEL
LIN {X 0,Y 403.27,Z 599.415,A -85,B 0,C 180,E1 -10784.846,E2 -10784.846} C_VEL
LIN {X 0,Y 403.708,Z 594.302,A -85,B 0,C 180,E1 -10786.407,E2 -10786.407} C_VEL
LIN {X 0,Y 404.215,Z 587.829,A -85,B 0,C 180,E1 -10787.957,E2 -10787.957} C_VEL
LIN {X 0,Y 404.875,Z 579.729,A -85,B 0,C 180,E1 -10789.498,E2 -10789.498} C_VEL
LIN {X 0,Y 405.67,Z 570.44,A -85,B 0,C 180,E1 -10790.917,E2 -10790.917} C_VEL
LIN {X 0,Y 406.496,Z 560.13,A -85,B 0,C 180,E1 -10792.175,E2 -10792.175} C_VEL
LIN {X 0,Y 407.312,Z 549.858,A -85,B 0,C 180,E1 -10793.187,E2 -10793.187} C_VEL
LIN {X 0,Y 408.012,Z 538.708,A -85,B 0,C 180,E1 -10794.068,E2 -10794.068} C_VEL
LIN {X 0,Y 408.698,Z 526.259,A -85,B 0,C 180,E1 -10794.82,E2 -10794.82} C_VEL
LIN {X 0,Y 409.236,Z 513.174,A -85,B 0,C 180,E1 -10795.395,E2 -10795.395} C_VEL
LIN {X 0,Y 409.648,Z 499.187,A -85,B 0,C 180,E1 -10795.777,E2 -10795.777} C_VEL
LIN {X 0,Y 411.311,Z 419.391,A -85,B 0,C 180,E1 -10797.433,E2 -10797.433} C_VEL
LIN {X 0,Y 408.231,Z 404.335,A -85,B 0,C 180,E1 -10797.968,E2 -10797.968} C_VEL
LIN {X 0,Y 406.644,Z 397.467,A -85,B 0,C 180,E1 -10798.242,E2 -10798.242} C_VEL
LIN {X 0,Y 406.563,Z 391.434,A -85,B 0,C 180,E1 -10799.505,E2 -10799.505} C_VEL
LIN {X 0,Y 404.716,Z 382.413,A -85,B 0,C 180,E1 -10801.493,E2 -10801.493} C_VEL
LIN {X 0,Y 404.47,Z 381.105,A -85,B 0,C 180,E1 -10801.805,E2 -10801.805} C_VEL
LIN {X 0,Y 404.413,Z 381.114,A -85,B 0,C 180,E1 -10805.985,E2 -10805.985} C_VEL
LIN {X 0,Y 404.412,Z 381.111,A -85,B 0,C 180,E1 -10807.991,E2 -10807.991} C_VEL
LIN {X 0,Y 404.259,Z 381.129,A -85,B 0,C 180,E1 -10812.041,E2 -10812.041} C_VEL
LIN {X 0,Y 404.202,Z 381.136,A -85,B 0,C 180,E1 -10815.118,E2 -10815.118} C_VEL
LIN {X 0,Y 404.204,Z 381.137,A -85,B 0,C 180,E1 -10818.238,E2 -10818.238} C_VEL
LIN {X 0,Y 404.191,Z 381.137,A -85,B 0,C 180,E1 -10821.416,E2 -10821.416} C_VEL
LIN {X 0,Y 404.169,Z 381.138,A -85,B 0,C 180,E1 -10824.666,E2 -10824.666} C_VEL
LIN {X 0,Y 404.188,Z 381.138,A -85,B 0,C 180,E1 -10828,E2 -10828} C_VEL
LIN {X 0,Y 404.138,Z 381.145,A -85,B 0,C 180,E1 -10831.561,E2 -10831.561} C_VEL
LIN {X 0,Y 404.177,Z 381.139,A -85,B 0,C 180,E1 -10835.017,E2 -10835.017} C_VEL
LIN {X 0,Y 404.151,Z 381.141,A -85,B 0,C 180,E1 -10838.757,E2 -10838.757} C_VEL
LIN {X 0,Y 404.117,Z 381.148,A -85,B 0,C 180,E1 -10841.601,E2 -10841.601} C_VEL
LIN {X 0,Y 404.143,Z 381.14,A -85,B 0,C 180,E1 -10844.524,E2 -10844.524} C_VEL
LIN {X 0,Y 404.133,Z 381.145,A -85,B 0,C 180,E1 -10847.297,E2 -10847.297} C_VEL
LIN {X 0,Y 404.163,Z 381.139,A -85,B 0,C 180,E1 -10849.957,E2 -10849.957} C_VEL
LIN {X 0,Y 404.135,Z 381.146,A -85,B 0,C 180,E1 -10853.126,E2 -10853.126} C_VEL
LIN {X 0,Y 404.141,Z 381.143,A -85,B 0,C 180,E1 -10856.189,E2 -10856.189} C_VEL
LIN {X 0,Y 404.153,Z 381.142,A -85,B 0,C 180,E1 -10859.717,E2 -10859.717} C_VEL
LIN {X 0,Y 404.263,Z 381.179,A -85,B 0,C 180,E1 -10862.139,E2 -10862.139} C_VEL
LIN {X 0,Y 406.659,Z 393.35,A -85,B 0,C 180,E1 -10864.951,E2 -10864.951} C_VEL
LIN {X 0,Y 407.277,Z 398.732,A -85,B 0,C 180,E1 -10866.145,E2 -10866.145} C_VEL
LIN {X 0,Y 406.144,Z 414.48,A -85,B 0,C 180,E1 -10869.431,E2 -10869.431} C_VEL
LIN {X 0,Y 405.946,Z 417.371,A -85,B 0,C 180,E1 -10870.028,E2 -10870.028} C_VEL
LIN {X 0,Y 408.884,Z 435.242,A -85,B 0,C 180,E1 -10870.631,E2 -10870.631} C_VEL
LIN {X 0,Y 410.333,Z 446.787,A -85,B 0,C 180,E1 -10870.981,E2 -10870.981} C_VEL
LIN {X 0,Y 409.202,Z 506.509,A -85,B 0,C 180,E1 -10872.22,E2 -10872.22} C_VEL
LIN {X 0,Y 408.864,Z 528.77,A -85,B 0,C 180,E1 -10872.657,E2 -10872.657} C_VEL
LIN {X 0,Y 408.273,Z 542.077,A -85,B 0,C 180,E1 -10873.114,E2 -10873.114} C_VEL
LIN {X 0,Y 407.669,Z 554.366,A -85,B 0,C 180,E1 -10873.733,E2 -10873.733} C_VEL
LIN {X 0,Y 406.919,Z 565.358,A -85,B 0,C 180,E1 -10874.474,E2 -10874.474} C_VEL
LIN {X 0,Y 406.112,Z 576.92,A -85,B 0,C 180,E1 -10875.469,E2 -10875.469} C_VEL
LIN {X 0,Y 405.391,Z 587.361,A -85,B 0,C 180,E1 -10876.598,E2 -10876.598} C_VEL
LIN {X 0,Y 404.796,Z 595.84,A -85,B 0,C 180,E1 -10877.722,E2 -10877.722} C_VEL
LIN {X 0,Y 404.012,Z 605.048,A -85,B 0,C 180,E1 -10879.224,E2 -10879.224} C_VEL
LIN {X 0,Y 403.52,Z 612.463,A -85,B 0,C 180,E1 -10880.73,E2 -10880.73} C_VEL
LIN {X 0,Y 403.234,Z 617.488,A -85,B 0,C 180,E1 -10881.986,E2 -10881.986} C_VEL
LIN {X 0,Y 402.978,Z 623.149,A -85,B 0,C 180,E1 -10883.769,E2 -10883.769} C_VEL
LIN {X 0,Y 402.932,Z 626.09,A -85,B 0,C 180,E1 -10884.998,E2 -10884.998} C_VEL
LIN {X 0,Y 402.852,Z 628.011,A -85,B 0,C 180,E1 -10886,E2 -10886} C_VEL
LIN {X 0,Y 402.825,Z 629.485,A -85,B 0,C 180,E1 -10887.001,E2 -10887.001} C_VEL
LIN {X 0,Y 402.864,Z 630.519,A -85,B 0,C 180,E1 -10888.002,E2 -10888.002} C_VEL
LIN {X 0,Y 402.862,Z 631.157,A -85,B 0,C 180,E1 -10889.002,E2 -10889.002} C_VEL
LIN {X 0,Y 402.851,Z 631.403,A -85,B 0,C 180,E1 -10890.001,E2 -10890.001} C_VEL
LIN {X 0,Y 402.862,Z 631.228,A -85,B 0,C 180,E1 -10891.001,E2 -10891.001} C_VEL
LIN {X 0,Y 402.865,Z 630.631,A -85,B 0,C 180,E1 -10892.001,E2 -10892.001} C_VEL
LIN {X 0,Y 402.853,Z 628.25,A -85,B 0,C 180,E1 -10894.003,E2 -10894.003} C_VEL
LIN {X 0,Y 402.919,Z 625.317,A -85,B 0,C 180,E1 -10895.506,E2 -10895.506} C_VEL
LIN {X 0,Y 403.081,Z 621.344,A -85,B 0,C 180,E1 -10897.012,E2 -10897.012} C_VEL
LIN {X 0,Y 403.422,Z 615.244,A -85,B 0,C 180,E1 -10898.769,E2 -10898.769} C_VEL
LIN {X 0,Y 403.908,Z 608.561,A -85,B 0,C 180,E1 -10900.275,E2 -10900.275} C_VEL
LIN {X 0,Y 404.557,Z 600.269,A -85,B 0,C 180,E1 -10901.779,E2 -10901.779} C_VEL
LIN {X 0,Y 405.312,Z 591.798,A -85,B 0,C 180,E1 -10903.029,E2 -10903.029} C_VEL
LIN {X 0,Y 405.982,Z 582.062,A -85,B 0,C 180,E1 -10904.205,E2 -10904.205} C_VEL
LIN {X 0,Y 406.862,Z 571.022,A -85,B 0,C 180,E1 -10905.274,E2 -10905.274} C_VEL
LIN {X 0,Y 407.705,Z 559.747,A -85,B 0,C 180,E1 -10906.14,E2 -10906.14} C_VEL
LIN {X 0,Y 408.462,Z 547.082,A -85,B 0,C 180,E1 -10906.88,E2 -10906.88} C_VEL
LIN {X 0,Y 409.127,Z 533.617,A -85,B 0,C 180,E1 -10907.431,E2 -10907.431} C_VEL
LIN {X 0,Y 409.624,Z 520.276,A -85,B 0,C 180,E1 -10907.764,E2 -10907.764} C_VEL
LIN {X 0,Y 410.559,Z 445.93,A -85,B 0,C 180,E1 -10909.143,E2 -10909.143} C_VEL
LIN {X 0,Y 406.351,Z 420.387,A -85,B 0,C 180,E1 -10909.866,E2 -10909.866} C_VEL
LIN {X 0,Y 406.06,Z 418.379,A -85,B 0,C 180,E1 -10909.963,E2 -10909.963} C_VEL
LIN {X 0,Y 407.518,Z 400.245,A -85,B 0,C 180,E1 -10913.787,E2 -10913.787} C_VEL
LIN {X 0,Y 407.462,Z 397.213,A -85,B 0,C 180,E1 -10914.455,E2 -10914.455} C_VEL
LIN {X 0,Y 405.168,Z 385.499,A -85,B 0,C 180,E1 -10917.233,E2 -10917.233} C_VEL
LIN {X 0,Y 404.214,Z 381.14,A -85,B 0,C 180,E1 -10918.353,E2 -10918.353} C_VEL
LIN {X 0,Y 404.145,Z 381.147,A -85,B 0,C 180,E1 -10921.559,E2 -10921.559} C_VEL
LIN {X 0,Y 404.19,Z 381.14,A -85,B 0,C 180,E1 -10925.017,E2 -10925.017} C_VEL
LIN {X 0,Y 404.161,Z 381.144,A -85,B 0,C 180,E1 -10928.757,E2 -10928.757} C_VEL
LIN {X 0,Y 404.129,Z 381.148,A -85,B 0,C 180,E1 -10931.6,E2 -10931.6} C_VEL
LIN {X 0,Y 404.151,Z 381.144,A -85,B 0,C 180,E1 -10934.523,E2 -10934.523} C_VEL
LIN {X 0,Y 404.142,Z 381.143,A -85,B 0,C 180,E1 -10937.296,E2 -10937.296} C_VEL
LIN {X 0,Y 404.174,Z 381.133,A -85,B 0,C 180,E1 -10939.956,E2 -10939.956} C_VEL
LIN {X 0,Y 404.141,Z 381.142,A -85,B 0,C 180,E1 -10943.126,E2 -10943.126} C_VEL
LIN {X 0,Y 404.15,Z 381.138,A -85,B 0,C 180,E1 -10946.188,E2 -10946.188} C_VEL
LIN {X 0,Y 404.151,Z 381.133,A -85,B 0,C 180,E1 -10949.715,E2 -10949.715} C_VEL
LIN {X 0,Y 404.201,Z 381.129,A -85,B 0,C 180,E1 -10953.123,E2 -10953.123} C_VEL
LIN {X 0,Y 404.182,Z 381.136,A -85,B 0,C 180,E1 -10955.335,E2 -10955.335} C_VEL
LIN {X 0,Y 404.166,Z 381.141,A -85,B 0,C 180,E1 -10958.582,E2 -10958.582} C_VEL
LIN {X 0,Y 404.216,Z 381.126,A -85,B 0,C 180,E1 -10961.762,E2 -10961.762} C_VEL
LIN {X 0,Y 404.212,Z 381.127,A -85,B 0,C 180,E1 -10964.882,E2 -10964.882} C_VEL
LIN {X 0,Y 404.262,Z 381.129,A -85,B 0,C 180,E1 -10967.959,E2 -10967.959} C_VEL
LIN {X 0,Y 404.44,Z 381.108,A -85,B 0,C 180,E1 -10972.1,E2 -10972.1} C_VEL
LIN {X 0,Y 404.43,Z 381.103,A -85,B 0,C 180,E1 -10974.015,E2 -10974.015} C_VEL
LIN {X 0,Y 404.486,Z 381.098,A -85,B 0,C 180,E1 -10978.009,E2 -10978.009} C_VEL
LIN {X 0,Y 404.616,Z 381.083,A -85,B 0,C 180,E1 -10980,E2 -10980} C_VEL
LIN {X 0,Y 404.422,Z 381.105,A -85,B 0,C 180,E1 -10982.988,E2 -10982.988} C_VEL
LIN {X 0,Y 404.418,Z 381.104,A -85,B 0,C 180,E1 -10986.987,E2 -10986.987} C_VEL
LIN {X 0,Y 404.265,Z 381.13,A -85,B 0,C 180,E1 -10990.012,E2 -10990.012} C_VEL
LIN {X 0,Y 404.273,Z 381.127,A -85,B 0,C 180,E1 -10993.211,E2 -10993.211} C_VEL
LIN {X 0,Y 404.222,Z 381.133,A -85,B 0,C 180,E1 -10997.007,E2 -10997.007} C_VEL
LIN {X 0,Y 404.17,Z 381.14,A -85,B 0,C 180,E1 -11000.351,E2 -11000.351} C_VEL
LIN {X 0,Y 404.175,Z 381.138,A -85,B 0,C 180,E1 -11003.574,E2 -11003.574} C_VEL
LIN {X 0,Y 404.204,Z 381.137,A -85,B 0,C 180,E1 -11006.877,E2 -11006.877} C_VEL
LIN {X 0,Y 404.269,Z 381.274,A -85,B 0,C 180,E1 -11007.548,E2 -11007.548} C_VEL
LIN {X 0,Y 406.093,Z 390.699,A -85,B 0,C 180,E1 -11010.125,E2 -11010.125} C_VEL
LIN {X 0,Y 406.67,Z 394.887,A -85,B 0,C 180,E1 -11011.229,E2 -11011.229} C_VEL
LIN {X 0,Y 406.478,Z 398.725,A -85,B 0,C 180,E1 -11012.169,E2 -11012.169} C_VEL
LIN {X 0,Y 410.916,Z 419.622,A -85,B 0,C 180,E1 -11012.821,E2 -11012.821} C_VEL
LIN {X 0,Y 409.55,Z 505.677,A -85,B 0,C 180,E1 -11014.434,E2 -11014.434} C_VEL
LIN {X 0,Y 409.067,Z 519.247,A -85,B 0,C 180,E1 -11014.892,E2 -11014.892} C_VEL
LIN {X 0,Y 408.48,Z 532.278,A -85,B 0,C 180,E1 -11015.551,E2 -11015.551} C_VEL
LIN {X 0,Y 407.76,Z 543.937,A -85,B 0,C 180,E1 -11016.353,E2 -11016.353} C_VEL
LIN {X 0,Y 406.905,Z 555.679,A -85,B 0,C 180,E1 -11017.39,E2 -11017.39} C_VEL
LIN {X 0,Y 406.076,Z 566.007,A -85,B 0,C 180,E1 -11018.54,E2 -11018.54} C_VEL
LIN {X 0,Y 405.166,Z 575.977,A -85,B 0,C 180,E1 -11019.927,E2 -11019.927} C_VEL
LIN {X 0,Y 404.501,Z 584.05,A -85,B 0,C 180,E1 -11021.318,E2 -11021.318} C_VEL
LIN {X 0,Y 403.975,Z 590.688,A -85,B 0,C 180,E1 -11022.726,E2 -11022.726} C_VEL
LIN {X 0,Y 403.467,Z 597.003,A -85,B 0,C 180,E1 -11024.423,E2 -11024.423} C_VEL
LIN {X 0,Y 403.213,Z 601.014,A -85,B 0,C 180,E1 -11025.796,E2 -11025.796} C_VEL
LIN {X 0,Y 402.96,Z 604.074,A -85,B 0,C 180,E1 -11027.14,E2 -11027.14} C_VEL
LIN {X 0,Y 402.794,Z 606.485,A -85,B 0,C 180,E1 -11028.614,E2 -11028.614} C_VEL
LIN {X 0,Y 402.695,Z 608.053,A -85,B 0,C 180,E1 -11030.167,E2 -11030.167} C_VEL
LIN {X 0,Y 402.661,Z 608.656,A -85,B 0,C 180,E1 -11031.76,E2 -11031.76} C_VEL
LIN {X 0,Y 402.677,Z 608.105,A -85,B 0,C 180,E1 -11033.599,E2 -11033.599} C_VEL
LIN {X 0,Y 402.752,Z 606.635,A -85,B 0,C 180,E1 -11035.1,E2 -11035.1} C_VEL
LIN {X 0,Y 402.967,Z 603.741,A -85,B 0,C 180,E1 -11036.841,E2 -11036.841} C_VEL
LIN {X 0,Y 403.258,Z 599.302,A -85,B 0,C 180,E1 -11038.647,E2 -11038.647} C_VEL
LIN {X 0,Y 403.536,Z 594.473,A -85,B 0,C 180,E1 -11040.126,E2 -11040.126} C_VEL
LIN {X 0,Y 404.018,Z 587.959,A -85,B 0,C 180,E1 -11041.703,E2 -11041.703} C_VEL
LIN {X 0,Y 404.592,Z 580.477,A -85,B 0,C 180,E1 -11043.15,E2 -11043.15} C_VEL
LIN {X 0,Y 405.213,Z 572.502,A -85,B 0,C 180,E1 -11044.408,E2 -11044.408} C_VEL
LIN {X 0,Y 406.015,Z 562.393,A -85,B 0,C 180,E1 -11045.704,E2 -11045.704} C_VEL
LIN {X 0,Y 406.825,Z 551.182,A -85,B 0,C 180,E1 -11046.857,E2 -11046.857} C_VEL
LIN {X 0,Y 407.456,Z 540.882,A -85,B 0,C 180,E1 -11047.698,E2 -11047.698} C_VEL
LIN {X 0,Y 408.053,Z 529.227,A -85,B 0,C 180,E1 -11048.444,E2 -11048.444} C_VEL
LIN {X 0,Y 408.649,Z 516.133,A -85,B 0,C 180,E1 -11049.058,E2 -11049.058} C_VEL
LIN {X 0,Y 409.037,Z 503.012,A -85,B 0,C 180,E1 -11049.457,E2 -11049.457} C_VEL
LIN {X 0,Y 410.172,Z 419.154,A -85,B 0,C 180,E1 -11051,E2 -11051} C_VEL
LIN {X 0,Y 406.045,Z 397.865,A -85,B 0,C 180,E1 -11051.618,E2 -11051.618} C_VEL
LIN {X 0,Y 406.284,Z 392.575,A -85,B 0,C 180,E1 -11052.897,E2 -11052.897} C_VEL
LIN {X 0,Y 405.847,Z 389.804,A -85,B 0,C 180,E1 -11053.605,E2 -11053.605} C_VEL
LIN {X 0,Y 404.777,Z 388.239,A -85,B 0,C 180,E1 -11054.082,E2 -11054.082} C_VEL
LIN {X 0,Y 397.973,Z 383.762,A -85,B 0,C 180,E1 -11055.598,E2 -11055.598} C_VEL
LIN {X 0,Y 397.222,Z 382.008,A -85,B 0,C 180,E1 -11056.152,E2 -11056.152} C_VEL
LIN {X 0,Y 397.223,Z 382.002,A -85,B 0,C 180,E1 -11059.808,E2 -11059.808} C_VEL
LIN {X 0,Y 397.323,Z 381.991,A -85,B 0,C 180,E1 -11062.886,E2 -11062.886} C_VEL
LIN {X 0,Y 397.252,Z 382,A -85,B 0,C 180,E1 -11064.924,E2 -11064.924} C_VEL
LIN {X 0,Y 397.454,Z 381.975,A -85,B 0,C 180,E1 -11067.972,E2 -11067.972} C_VEL
LIN {X 0,Y 397.583,Z 381.96,A -85,B 0,C 180,E1 -11069.999,E2 -11069.999} C_VEL
LIN {X 0,Y 397.384,Z 381.982,A -85,B 0,C 180,E1 -11073.04,E2 -11073.04} C_VEL
LIN {X 0,Y 397.367,Z 381.983,A -85,B 0,C 180,E1 -11077.11,E2 -11077.11} C_VEL
LIN {X 0,Y 397.219,Z 382.008,A -85,B 0,C 180,E1 -11080.19,E2 -11080.19} C_VEL
LIN {X 0,Y 397.228,Z 382.001,A -85,B 0,C 180,E1 -11083.32,E2 -11083.32} C_VEL
LIN {X 0,Y 397.172,Z 382.01,A -85,B 0,C 180,E1 -11086.445,E2 -11086.445} C_VEL
LIN {X 0,Y 397.148,Z 382.014,A -85,B 0,C 180,E1 -11089.646,E2 -11089.646} C_VEL
LIN {X 0,Y 397.11,Z 382.015,A -85,B 0,C 180,E1 -11093.031,E2 -11093.031} C_VEL
LIN {X 0,Y 397.133,Z 382.015,A -85,B 0,C 180,E1 -11096.257,E2 -11096.257} C_VEL
LIN {X 0,Y 397.124,Z 382.014,A -85,B 0,C 180,E1 -11098.542,E2 -11098.542} C_VEL
LIN {X 0,Y 397.108,Z 382.019,A -85,B 0,C 180,E1 -11102.067,E2 -11102.067} C_VEL
LIN {X 0,Y 397.116,Z 382.02,A -85,B 0,C 180,E1 -11105.502,E2 -11105.502} C_VEL
LIN {X 0,Y 397.133,Z 382.013,A -85,B 0,C 180,E1 -11108.861,E2 -11108.861} C_VEL
LIN {X 0,Y 397.11,Z 382.016,A -85,B 0,C 180,E1 -11112.259,E2 -11112.259} C_VEL
LIN {X 0,Y 397.163,Z 382.045,A -85,B 0,C 180,E1 -11115.19,E2 -11115.19} C_VEL
LIN {X 0,Y 398.826,Z 391.511,A -85,B 0,C 180,E1 -11117.274,E2 -11117.274} C_VEL
LIN {X 0,Y 398.807,Z 396.908,A -85,B 0,C 180,E1 -11118.381,E2 -11118.381} C_VEL
LIN {X 0,Y 402.898,Z 419.355,A -85,B 0,C 180,E1 -11119.039,E2 -11119.039} C_VEL
LIN {X 0,Y 401.385,Z 505.917,A -85,B 0,C 180,E1 -11120.806,E2 -11120.806} C_VEL
LIN {X 0,Y 400.937,Z 519.146,A -85,B 0,C 180,E1 -11121.276,E2 -11121.276} C_VEL
LIN {X 0,Y 400.388,Z 531.762,A -85,B 0,C 180,E1 -11121.935,E2 -11121.935} C_VEL
LIN {X 0,Y 399.835,Z 542.459,A -85,B 0,C 180,E1 -11122.669,E2 -11122.669} C_VEL
LIN {X 0,Y 399.158,Z 553.5,A -85,B 0,C 180,E1 -11123.623,E2 -11123.623} C_VEL
LIN {X 0,Y 398.394,Z 564.817,A -85,B 0,C 180,E1 -11124.863,E2 -11124.863} C_VEL
LIN {X 0,Y 397.695,Z 574.354,A -85,B 0,C 180,E1 -11126.155,E2 -11126.155} C_VEL
LIN {X 0,Y 397.119,Z 583.098,A -85,B 0,C 180,E1 -11127.632,E2 -11127.632} C_VEL
LIN {X 0,Y 396.606,Z 590.042,A -85,B 0,C 180,E1 -11129.076,E2 -11129.076} C_VEL
LIN {X 0,Y 396.306,Z 594.985,A -85,B 0,C 180,E1 -11130.334,E2 -11130.334} C_VEL
LIN {X 0,Y 396.013,Z 600.073,A -85,B 0,C 180,E1 -11131.946,E2 -11131.946} C_VEL
LIN {X 0,Y 395.821,Z 604.076,A -85,B 0,C 180,E1 -11133.648,E2 -11133.648} C_VEL
LIN {X 0,Y 395.709,Z 606.199,A -85,B 0,C 180,E1 -11134.925,E2 -11134.925} C_VEL
LIN {X 0,Y 395.603,Z 607.376,A -85,B 0,C 180,E1 -11135.883,E2 -11135.883} C_VEL
LIN {X 0,Y 395.56,Z 608.488,A -85,B 0,C 180,E1 -11137.497,E2 -11137.497} C_VEL
LIN {X 0,Y 395.562,Z 608.52,A -85,B 0,C 180,E1 -11139.185,E2 -11139.185} C_VEL
LIN {X 0,Y 395.654,Z 607.898,A -85,B 0,C 180,E1 -11140.289,E2 -11140.289} C_VEL
LIN {X 0,Y 395.717,Z 606.87,A -85,B 0,C 180,E1 -11141.356,E2 -11141.356} C_VEL
LIN {X 0,Y 395.84,Z 605.335,A -85,B 0,C 180,E1 -11142.432,E2 -11142.432} C_VEL
LIN {X 0,Y 396.081,Z 602.134,A -85,B 0,C 180,E1 -11144.036,E2 -11144.036} C_VEL
LIN {X 0,Y 396.397,Z 597.79,A -85,B 0,C 180,E1 -11145.628,E2 -11145.628} C_VEL
LIN {X 0,Y 396.936,Z 591.705,A -85,B 0,C 180,E1 -11147.331,E2 -11147.331} C_VEL
LIN {X 0,Y 397.505,Z 585.116,A -85,B 0,C 180,E1 -11148.785,E2 -11148.785} C_VEL
LIN {X 0,Y 398.257,Z 576.272,A -85,B 0,C 180,E1 -11150.349,E2 -11150.349} C_VEL
LIN {X 0,Y 399.097,Z 567.035,A -85,B 0,C 180,E1 -11151.666,E2 -11151.666} C_VEL
LIN {X 0,Y 400.031,Z 555.857,A -85,B 0,C 180,E1 -11152.936,E2 -11152.936} C_VEL
LIN {X 0,Y 400.886,Z 544.573,A -85,B 0,C 180,E1 -11153.962,E2 -11153.962} C_VEL
LIN {X 0,Y 401.718,Z 531.757,A -85,B 0,C 180,E1 -11154.856,E2 -11154.856} C_VEL
LIN {X 0,Y 402.381,Z 518.802,A -85,B 0,C 180,E1 -11155.527,E2 -11155.527} C_VEL
LIN {X 0,Y 402.869,Z 505.12,A -85,B 0,C 180,E1 -11155.999,E2 -11155.999} C_VEL
LIN {X 0,Y 404.816,Z 420.662,A -85,B 0,C 180,E1 -11157.803,E2 -11157.803} C_VEL
LIN {X 0,Y 401.531,Z 404.446,A -85,B 0,C 180,E1 -11158.402,E2 -11158.402} C_VEL
LIN {X 0,Y 399.898,Z 397.597,A -85,B 0,C 180,E1 -11158.707,E2 -11158.707} C_VEL
LIN {X 0,Y 399.677,Z 392.741,A -85,B 0,C 180,E1 -11159.748,E2 -11159.748} C_VEL
LIN {X 0,Y 397.822,Z 383.677,A -85,B 0,C 180,E1 -11161.772,E2 -11161.772} C_VEL
LIN {X 0,Y 397.409,Z 381.986,A -85,B 0,C 180,E1 -11162.217,E2 -11162.217} C_VEL
LIN {X 0,Y 397.365,Z 381.992,A -85,B 0,C 180,E1 -11166.092,E2 -11166.092} C_VEL
LIN {X 0,Y 397.366,Z 381.988,A -85,B 0,C 180,E1 -11168.134,E2 -11168.134} C_VEL
LIN {X 0,Y 397.219,Z 382.005,A -85,B 0,C 180,E1 -11172.258,E2 -11172.258} C_VEL
LIN {X 0,Y 397.174,Z 382.012,A -85,B 0,C 180,E1 -11175.392,E2 -11175.392} C_VEL
LIN {X 0,Y 397.161,Z 382.014,A -85,B 0,C 180,E1 -11178.573,E2 -11178.573} C_VEL
LIN {X 0,Y 397.167,Z 382.014,A -85,B 0,C 180,E1 -11181.814,E2 -11181.814} C_VEL
LIN {X 0,Y 397.144,Z 382.016,A -85,B 0,C 180,E1 -11185.514,E2 -11185.514} C_VEL
LIN {X 0,Y 397.117,Z 382.017,A -85,B 0,C 180,E1 -11188.544,E2 -11188.544} C_VEL
LIN {X 0,Y 397.102,Z 382.021,A -85,B 0,C 180,E1 -11192.069,E2 -11192.069} C_VEL
LIN {X 0,Y 397.111,Z 382.02,A -85,B 0,C 180,E1 -11195.505,E2 -11195.505} C_VEL
LIN {X 0,Y 397.125,Z 382.017,A -85,B 0,C 180,E1 -11198.863,E2 -11198.863} C_VEL
LIN {X 0,Y 397.064,Z 382.023,A -85,B 0,C 180,E1 -11202.268,E2 -11202.268} C_VEL
LIN {X 0,Y 397.085,Z 382.024,A -85,B 0,C 180,E1 -11205.069,E2 -11205.069} C_VEL
LIN {X 0,Y 397.062,Z 382.023,A -85,B 0,C 180,E1 -11208.022,E2 -11208.022} C_VEL
LIN {X 0,Y 397.127,Z 382.018,A -85,B 0,C 180,E1 -11211.139,E2 -11211.139} C_VEL
LIN {X 0,Y 397.115,Z 382.019,A -85,B 0,C 180,E1 -11214.498,E2 -11214.498} C_VEL
LIN {X 0,Y 397.108,Z 382.018,A -85,B 0,C 180,E1 -11217.933,E2 -11217.933} C_VEL
LIN {X 0,Y 397.217,Z 382.074,A -85,B 0,C 180,E1 -11221.877,E2 -11221.877} C_VEL
LIN {X 0,Y 399.623,Z 394.304,A -85,B 0,C 180,E1 -11224.758,E2 -11224.758} C_VEL
LIN {X 0,Y 400.375,Z 399.29,A -85,B 0,C 180,E1 -11225.893,E2 -11225.893} C_VEL
LIN {X 0,Y 399.226,Z 414.119,A -85,B 0,C 180,E1 -11229.046,E2 -11229.046} C_VEL
LIN {X 0,Y 399.079,Z 416.57,A -85,B 0,C 180,E1 -11229.564,E2 -11229.564} C_VEL
LIN {X 0,Y 402.443,Z 436.773,A -85,B 0,C 180,E1 -11230.274,E2 -11230.274} C_VEL
LIN {X 0,Y 403.773,Z 448.143,A -85,B 0,C 180,E1 -11230.624,E2 -11230.624} C_VEL
LIN {X 0,Y 402.048,Z 528.832,A -85,B 0,C 180,E1 -11232.386,E2 -11232.386} C_VEL
LIN {X 0,Y 401.456,Z 541.205,A -85,B 0,C 180,E1 -11232.819,E2 -11232.819} C_VEL
LIN {X 0,Y 400.833,Z 553.719,A -85,B 0,C 180,E1 -11233.447,E2 -11233.447} C_VEL
LIN {X 0,Y 400.053,Z 564.794,A -85,B 0,C 180,E1 -11234.2,E2 -11234.2} C_VEL
LIN {X 0,Y 399.325,Z 575.142,A -85,B 0,C 180,E1 -11235.086,E2 -11235.086} C_VEL
LIN {X 0,Y 398.514,Z 586.346,A -85,B 0,C 180,E1 -11236.291,E2 -11236.291} C_VEL
LIN {X 0,Y 397.837,Z 595.459,A -85,B 0,C 180,E1 -11237.504,E2 -11237.504} C_VEL
LIN {X 0,Y 397.009,Z 604.71,A -85,B 0,C 180,E1 -11239.031,E2 -11239.031} C_VEL
LIN {X 0,Y 396.491,Z 612.151,A -85,B 0,C 180,E1 -11240.565,E2 -11240.565} C_VEL
LIN {X 0,Y 396.188,Z 617.2,A -85,B 0,C 180,E1 -11241.843,E2 -11241.843} C_VEL
LIN {X 0,Y 395.92,Z 622.091,A -85,B 0,C 180,E1 -11243.376,E2 -11243.376} C_VEL
LIN {X 0,Y 395.845,Z 625.84,A -85,B 0,C 180,E1 -11244.908,E2 -11244.908} C_VEL
LIN {X 0,Y 395.775,Z 627.77,A -85,B 0,C 180,E1 -11245.928,E2 -11245.928} C_VEL
LIN {X 0,Y 395.728,Z 629.259,A -85,B 0,C 180,E1 -11246.947,E2 -11246.947} C_VEL
LIN {X 0,Y 395.763,Z 630.301,A -85,B 0,C 180,E1 -11247.966,E2 -11247.966} C_VEL
LIN {X 0,Y 395.791,Z 630.947,A -85,B 0,C 180,E1 -11248.984,E2 -11248.984} C_VEL
LIN {X 0,Y 395.778,Z 631.199,A -85,B 0,C 180,E1 -11250.001,E2 -11250.001} C_VEL
LIN {X 0,Y 395.791,Z 631.037,A -85,B 0,C 180,E1 -11251.019,E2 -11251.019} C_VEL
LIN {X 0,Y 395.763,Z 630.444,A -85,B 0,C 180,E1 -11252.037,E2 -11252.037} C_VEL
LIN {X 0,Y 395.776,Z 628.074,A -85,B 0,C 180,E1 -11254.074,E2 -11254.074} C_VEL
LIN {X 0,Y 395.829,Z 624.701,A -85,B 0,C 180,E1 -11255.808,E2 -11255.808} C_VEL
LIN {X 0,Y 396.08,Z 619.608,A -85,B 0,C 180,E1 -11257.649,E2 -11257.649} C_VEL
LIN {X 0,Y 396.516,Z 613.06,A -85,B 0,C 180,E1 -11259.438,E2 -11259.438} C_VEL
LIN {X 0,Y 397.041,Z 605.883,A -85,B 0,C 180,E1 -11260.971,E2 -11260.971} C_VEL
LIN {X 0,Y 397.9,Z 596.953,A -85,B 0,C 180,E1 -11262.497,E2 -11262.497} C_VEL
LIN {X 0,Y 398.637,Z 588.159,A -85,B 0,C 180,E1 -11263.725,E2 -11263.725} C_VEL
LIN {X 0,Y 399.426,Z 578.12,A -85,B 0,C 180,E1 -11264.874,E2 -11264.874} C_VEL
LIN {X 0,Y 400.382,Z 566.562,A -85,B 0,C 180,E1 -11265.92,E2 -11265.92} C_VEL
LIN {X 0,Y 401.337,Z 554.059,A -85,B 0,C 180,E1 -11266.796,E2 -11266.796} C_VEL
LIN {X 0,Y 402.013,Z 541.342,A -85,B 0,C 180,E1 -11267.454,E2 -11267.454} C_VEL
LIN {X 0,Y 402.675,Z 527.941,A -85,B 0,C 180,E1 -11267.917,E2 -11267.917} C_VEL
LIN {X 0,Y 403.301,Z 490.376,A -85,B 0,C 180,E1 -11268.652,E2 -11268.652} C_VEL
LIN {X 0,Y 403.932,Z 447.028,A -85,B 0,C 180,E1 -11269.472,E2 -11269.472} C_VEL
